KUKA KRL program: Machining2.src

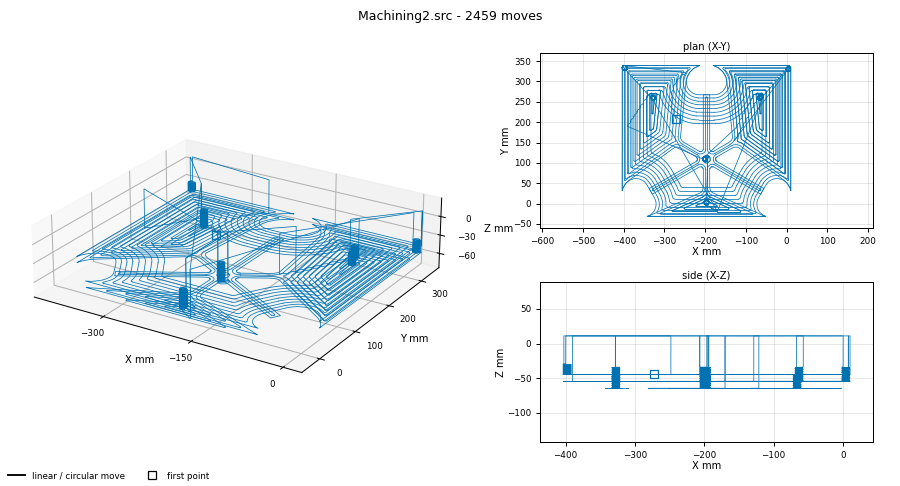
[picture p0: tool path of Machining2.src, 2459 of 2459 moves have a stored position in this frame; points joined in program order, loops and branches not executed]
&ACCESS RVP
&REL 1
&PARAM TEMPLATE = C:\KRC\Roboter\Template\vorgabe
&PARAM EDITMASK = *
DEF Machining2 ( )

; External program calls:
EXT Machining3()

CIRC {X -271.618,Y 203.851,Z -44.500,A 0.015,B -0.000,C -180.000},{X -272.375,Y 208.247,Z -44.500,A 0.015,B -0.000,C -180.000} C_DIS
CIRC {X -272.985,Y 212.625,Z -44.500,A 0.015,B 0.000,C 180.000},{X -275.736,Y 216.083,Z -44.500,A 0.015,B 0.000,C 180.000} C_DIS
CIRC {X -297.181,Y 237.599,Z -44.500,A 0.015,B -0.000,C 180.000},{X -311.042,Y 264.630,Z -44.500,A 0.015,B -0.000,C -180.000} C_DIS
CIRC {X -313.145,Y 267.504,Z -44.500,A 0.015,B 0.000,C 180.000},{X -316.534,Y 268.601,Z -44.500,A 0.015,B 0.000,C 180.000} C_DIS
LIN {X -329.332,Y 268.600,Z -44.500,A 0.015,B 0.000,C 180.000} C_DIS
CIRC {X -332.056,Y 267.472,Z -44.500,A 0.015,B 0.000,C -180.000},{X -333.185,Y 264.747,Z -44.500,A 0.015,B 0.000,C -180.000} C_DIS
LIN {X -333.181,Y 129.664,Z -44.500,A 0.015,B -0.000,C 180.000} C_DIS
CIRC {X -332.044,Y 125.846,Z -44.500,A 0.015,B 0.000,C 180.000},{X -329.005,Y 123.272,Z -44.500,A 0.015,B 0.000,C 180.000} C_DIS
CIRC {X -324.117,Y 121.053,Z -44.500,A 0.015,B 0.000,C 180.000},{X -319.285,Y 118.713,Z -44.500,A 0.015,B 0.000,C 180.000} C_DIS
CIRC {X -314.570,Y 116.140,Z -44.500,A 0.015,B 0.000,C -180.000},{X -310.050,Y 113.238,Z -44.500,A 0.015,B 0.000,C -180.000} C_DIS
CIRC {X -294.805,Y 99.946,Z -44.500,A 0.015,B 0.000,C -180.000},{X -282.838,Y 83.640,Z -44.500,A 0.015,B 0.000,C 180.000} C_DIS
LIN {X -263.188,Y 49.540,Z -44.500,A 0.015,B 0.000,C 180.000} C_DIS
CIRC {X -262.373,Y 48.033,Z -44.500,A 0.015,B 0.000,C 180.000},{X -261.642,Y 46.485,Z -44.500,A 0.015,B 0.000,C -180.000} C_DIS
CIRC {X -260.946,Y 44.921,Z -44.500,A 0.015,B 0.000,C 180.000},{X -260.238,Y 43.362,Z -44.500,A 0.015,B 0.000,C 180.000} C_DIS
CIRC {X -257.688,Y 40.428,Z -44.500,A 0.015,B 0.000,C -180.000},{X -253.958,Y 39.334,Z -44.500,A 0.015,B 0.000,C 180.000} C_DIS
LIN {X -139.525,Y 39.335,Z -44.500,A 0.015,B 0.000,C 180.000} C_DIS
CIRC {X -135.796,Y 40.433,Z -44.500,A 0.015,B -0.000,C -180.000},{X -133.257,Y 43.377,Z -44.500,A 0.015,B 0.000,C 180.000} C_DIS
CIRC {X -132.507,Y 45.047,Z -44.500,A 0.015,B 0.000,C 180.000},{X -131.768,Y 46.722,Z -44.500,A 0.015,B -0.000,C 180.000} C_DIS
CIRC {X -130.987,Y 48.379,Z -44.500,A 0.015,B 0.000,C -180.000},{X -130.115,Y 49.990,Z -44.500,A 0.015,B 0.000,C -180.000} C_DIS
LIN {X -109.644,Y 85.014,Z -44.500,A 0.015,B -0.000,C 180.000} C_DIS
CIRC {X -97.349,Y 101.310,Z -44.500,A 0.015,B 0.000,C 180.000},{X -81.729,Y 114.451,Z -44.500,A 0.015,B 0.000,C 180.000} C_DIS
CIRC {X -77.604,Y 116.999,Z -44.500,A 0.015,B 0.000,C 180.000},{X -73.317,Y 119.264,Z -44.500,A 0.015,B 0.000,C -180.000} C_DIS
CIRC {X -68.933,Y 121.328,Z -44.500,A 0.015,B 0.000,C -180.000},{X -64.497,Y 123.278,Z -44.500,A 0.015,B 0.000,C 180.000} C_DIS
CIRC {X -61.466,Y 125.799,Z -44.500,A 0.015,B 0.000,C 180.000},{X -60.330,Y 129.575,Z -44.500,A 0.015,B 0.000,C 180.000} C_DIS
LIN {X -60.333,Y 264.754,Z -44.500,A 0.015,B 0.000,C 180.000} C_DIS
CIRC {X -61.462,Y 267.478,Z -44.500,A 0.015,B 0.000,C 180.000},{X -64.186,Y 268.607,Z -44.500,A 0.015,B -0.000,C -180.000} C_DIS
LIN {X -76.977,Y 268.606,Z -44.500,A 0.015,B 0.000,C -180.000} C_DIS
CIRC {X -80.365,Y 267.510,Z -44.500,A 0.015,B 0.000,C 180.000},{X -82.468,Y 264.636,Z -44.500,A 0.015,B 0.000,C 180.000} C_DIS
CIRC {X -91.051,Y 245.836,Z -44.500,A 0.015,B 0.000,C -180.000},{X -103.514,Y 229.351,Z -44.500,A 0.015,B 0.000,C 180.000} C_DIS
CIRC {X -119.021,Y 215.739,Z -44.500,A 0.015,B -0.000,C -180.000},{X -136.787,Y 205.249,Z -44.500,A 0.015,B -0.000,C -180.000} C_DIS
CIRC {X -155.589,Y 198.757,Z -44.500,A 0.015,B 0.000,C 180.000},{X -175.343,Y 196.423,Z -44.500,A 0.015,B 0.000,C 180.000} C_DIS
LIN {X -214.895,Y 196.221,Z -44.500,A 0.015,B 0.000,C 180.000} C_DIS
CIRC {X -245.902,Y 200.993,Z -44.500,A 0.015,B 0.000,C 180.000},{X -274.038,Y 214.868,Z -44.500,A 0.015,B 0.000,C 180.000} C_DIS
CIRC {X -274.890,Y 215.471,Z -44.500,A 0.015,B 0.000,C 180.000},{X -275.736,Y 216.083,Z -44.500,A 0.015,B 0.000,C -180.000} C_DIS
CIRC {X -278.577,Y 219.932,Z -44.500,A 0.015,B 0.000,C 180.000},{X -278.721,Y 224.714,Z -44.500,A 0.015,B 0.000,C 180.000} C_DIS
CIRC {X -278.679,Y 229.444,Z -44.500,A 0.015,B 0.000,C 180.000},{X -281.022,Y 233.552,Z -44.500,A 0.015,B 0.000,C 180.000} C_DIS
CIRC {X -283.384,Y 236.013,Z -44.500,A 0.015,B 0.000,C -180.000},{X -285.659,Y 238.555,Z -44.500,A 0.015,B 0.000,C 180.000} C_DIS
CIRC {X -296.886,Y 255.155,Z -44.500,A 0.015,B 0.000,C 180.000},{X -303.914,Y 273.923,Z -44.500,A 0.015,B 0.000,C 180.000} C_DIS
CIRC {X -305.790,Y 276.833,Z -44.500,A 0.015,B 0.000,C -180.000},{X -309.063,Y 277.963,Z -44.500,A 0.015,B 0.000,C -180.000} C_DIS
LIN {X -338.695,Y 277.963,Z -44.500,A 0.015,B -0.000,C 180.000} C_DIS
CIRC {X -341.419,Y 276.834,Z -44.500,A 0.015,B -0.000,C -180.000},{X -342.547,Y 274.110,Z -44.500,A 0.015,B -0.000,C 180.000} C_DIS
LIN {X -342.543,Y 123.023,Z -44.500,A 0.015,B 0.000,C 180.000} C_DIS
CIRC {X -341.454,Y 119.492,Z -44.500,A 0.015,B 0.000,C 180.000},{X -338.566,Y 117.188,Z -44.500,A 0.015,B 0.000,C 180.000} C_DIS
CIRC {X -332.560,Y 114.714,Z -44.500,A 0.015,B 0.000,C 180.000},{X -326.639,Y 112.042,Z -44.500,A 0.015,B 0.000,C 180.000} C_DIS
CIRC {X -320.879,Y 109.028,Z -44.500,A 0.015,B 0.000,C -180.000},{X -315.388,Y 105.546,Z -44.500,A 0.015,B -0.000,C 180.000} C_DIS
CIRC {X -301.093,Y 93.048,Z -44.500,A 0.015,B 0.000,C -180.000},{X -289.921,Y 77.693,Z -44.500,A 0.015,B 0.000,C -180.000} C_DIS
LIN {X -271.167,Y 44.942,Z -44.500,A 0.015,B 0.000,C 180.000} C_DIS
CIRC {X -269.801,Y 42.329,Z -44.500,A 0.015,B 0.000,C 180.000},{X -268.653,Y 39.612,Z -44.500,A 0.015,B -0.000,C -180.000} C_DIS
CIRC {X -267.596,Y 36.862,Z -44.500,A 0.015,B 0.000,C 180.000},{X -266.491,Y 34.130,Z -44.500,A 0.015,B 0.000,C -180.000} C_DIS
CIRC {X -264.009,Y 31.107,Z -44.500,A 0.015,B 0.000,C 180.000},{X -260.265,Y 29.972,Z -44.500,A 0.015,B 0.000,C 180.000} C_DIS
LIN {X -133.256,Y 29.972,Z -44.500,A 0.015,B 0.000,C -180.000} C_DIS
CIRC {X -129.505,Y 31.106,Z -44.500,A 0.015,B -0.000,C -180.000},{X -127.010,Y 34.129,Z -44.500,A 0.015,B 0.000,C -180.000} C_DIS
CIRC {X -125.855,Y 36.970,Z -44.500,A 0.015,B 0.000,C 180.000},{X -124.756,Y 39.833,Z -44.500,A 0.015,B 0.000,C -180.000} C_DIS
CIRC {X -123.565,Y 42.662,Z -44.500,A 0.015,B 0.000,C -180.000},{X -122.142,Y 45.382,Z -44.500,A 0.015,B -0.000,C -180.000} C_DIS
LIN {X -103.037,Y 78.441,Z -44.500,A 0.015,B -0.000,C 180.000} C_DIS
CIRC {X -91.420,Y 94.078,Z -44.500,A 0.015,B 0.000,C 180.000},{X -76.544,Y 106.655,Z -44.500,A 0.015,B 0.000,C 180.000} C_DIS
CIRC {X -71.400,Y 109.776,Z -44.500,A 0.015,B 0.000,C 180.000},{X -66.016,Y 112.459,Z -44.500,A 0.015,B 0.000,C 180.000} C_DIS
CIRC {X -60.505,Y 114.859,Z -44.500,A 0.015,B 0.000,C -180.000},{X -54.946,Y 117.146,Z -44.500,A 0.015,B -0.000,C 180.000} C_DIS
CIRC {X -52.055,Y 119.473,Z -44.500,A 0.015,B 0.000,C -180.000},{X -50.967,Y 123.022,Z -44.500,A 0.015,B 0.000,C 180.000} C_DIS
LIN {X -50.971,Y 274.117,Z -44.500,A 0.015,B 0.000,C 180.000} C_DIS
CIRC {X -52.100,Y 276.841,Z -44.500,A 0.015,B 0.000,C -180.000},{X -54.824,Y 277.969,Z -44.500,A 0.015,B 0.000,C -180.000} C_DIS
LIN {X -84.496,Y 277.969,Z -44.500,A 0.015,B -0.000,C -180.000} C_DIS
CIRC {X -87.755,Y 276.836,Z -44.500,A 0.015,B 0.000,C -180.000},{X -89.608,Y 273.925,Z -44.500,A 0.015,B 0.000,C 180.000} C_DIS
CIRC {X -106.660,Y 239.262,Z -44.500,A 0.015,B -0.000,C -180.000},{X -137.083,Y 215.457,Z -44.500,A 0.015,B -0.000,C -180.000} C_DIS
CIRC {X -147.019,Y 211.354,Z -44.500,A 0.015,B -0.000,C -180.000},{X -157.305,Y 208.228,Z -44.500,A 0.015,B 0.000,C 180.000} C_DIS
CIRC {X -167.879,Y 206.247,Z -44.500,A 0.015,B 0.000,C -180.000},{X -178.617,Y 205.584,Z -44.500,A 0.015,B 0.000,C 180.000} C_DIS
LIN {X -216.069,Y 205.584,Z -44.500,A 0.015,B 0.000,C -180.000} C_DIS
CIRC {X -235.574,Y 207.795,Z -44.500,A 0.015,B 0.000,C -180.000},{X -254.089,Y 214.317,Z -44.500,A 0.015,B 0.000,C 180.000} C_DIS
CIRC {X -268.368,Y 222.797,Z -44.500,A 0.015,B -0.000,C -180.000},{X -281.022,Y 233.552,Z -44.500,A 0.015,B 0.000,C 180.000} C_DIS
CIRC {X -283.064,Y 237.540,Z -44.500,A 0.015,B 0.000,C -180.000},{X -282.419,Y 241.973,Z -44.500,A 0.015,B 0.000,C 180.000} C_DIS
CIRC {X -281.599,Y 246.322,Z -44.500,A 0.015,B -0.000,C 180.000},{X -283.108,Y 250.482,Z -44.500,A 0.015,B 0.000,C 180.000} C_DIS
CIRC {X -285.499,Y 254.008,Z -44.500,A 0.015,B -0.000,C -180.000},{X -287.754,Y 257.623,Z -44.500,A 0.015,B 0.000,C 180.000} C_DIS
CIRC {X -291.877,Y 265.858,Z -44.500,A 0.015,B 0.000,C 180.000},{X -294.729,Y 274.615,Z -44.500,A 0.015,B 0.000,C -180.000} C_DIS
CIRC {X -295.216,Y 276.775,Z -44.500,A 0.015,B 0.000,C 180.000},{X -295.626,Y 278.952,Z -44.500,A 0.015,B 0.000,C -180.000} C_DIS
CIRC {X -296.025,Y 281.130,Z -44.500,A 0.015,B -0.000,C 180.000},{X -296.480,Y 283.297,Z -44.500,A 0.015,B 0.000,C 180.000} C_DIS
CIRC {X -298.286,Y 286.195,Z -44.500,A 0.015,B 0.000,C -180.000},{X -301.508,Y 287.326,Z -44.500,A 0.015,B -0.000,C 180.000} C_DIS
LIN {X -348.057,Y 287.325,Z -44.500,A 0.015,B 0.000,C -180.000} C_DIS
CIRC {X -350.782,Y 286.196,Z -44.500,A 0.015,B 0.000,C 180.000},{X -351.910,Y 283.472,Z -44.500,A 0.015,B 0.000,C -180.000} C_DIS
LIN {X -351.906,Y 115.520,Z -44.500,A 0.015,B 0.000,C -180.000} C_DIS
CIRC {X -350.817,Y 112.320,Z -44.500,A 0.015,B 0.000,C -180.000},{X -348.003,Y 110.446,Z -44.500,A 0.015,B -0.000,C -180.000} C_DIS
CIRC {X -338.196,Y 107.179,Z -44.500,A 0.015,B 0.000,C 180.000},{X -328.868,Y 102.725,Z -44.500,A 0.015,B -0.000,C -180.000} C_DIS
CIRC {X -320.144,Y 97.184,Z -44.500,A 0.015,B 0.000,C -180.000},{X -312.124,Y 90.665,Z -44.500,A 0.015,B 0.000,C -180.000} C_DIS
CIRC {X -307.860,Y 86.416,Z -44.500,A 0.015,B 0.000,C -180.000},{X -303.971,Y 81.821,Z -44.500,A 0.015,B 0.000,C -180.000} C_DIS
CIRC {X -300.448,Y 76.943,Z -44.500,A 0.015,B 0.000,C -180.000},{X -297.267,Y 71.835,Z -44.500,A 0.015,B 0.000,C -180.000} C_DIS
LIN {X -283.335,Y 47.658,Z -44.500,A 0.015,B 0.000,C -180.000} C_DIS
CIRC {X -277.503,Y 36.349,Z -44.500,A 0.015,B 0.000,C -180.000},{X -272.749,Y 24.546,Z -44.500,A 0.015,B -0.000,C -180.000} C_DIS
CIRC {X -270.603,Y 21.694,Z -44.500,A 0.015,B 0.000,C -180.000},{X -267.203,Y 20.609,Z -44.500,A 0.015,B -0.000,C 180.000} C_DIS
LIN {X -126.309,Y 20.609,Z -44.500,A 0.015,B 0.000,C 180.000} C_DIS
CIRC {X -122.909,Y 21.694,Z -44.500,A 0.015,B 0.000,C -180.000},{X -120.763,Y 24.546,Z -44.500,A 0.015,B 0.000,C -180.000} C_DIS
CIRC {X -115.935,Y 36.521,Z -44.500,A 0.015,B -0.000,C -180.000},{X -110.007,Y 47.991,Z -44.500,A 0.015,B -0.000,C -180.000} C_DIS
LIN {X -96.029,Y 72.178,Z -44.500,A 0.015,B 0.000,C 180.000} C_DIS
CIRC {X -90.459,Y 80.530,Z -44.500,A 0.015,B -0.000,C -180.000},{X -83.866,Y 88.100,Z -44.500,A 0.015,B 0.000,C 180.000} C_DIS
CIRC {X -76.453,Y 94.859,Z -44.500,A 0.015,B 0.000,C 180.000},{X -68.393,Y 100.832,Z -44.500,A 0.015,B 0.000,C 180.000} C_DIS
CIRC {X -63.022,Y 103.997,Z -44.500,A 0.015,B 0.000,C -180.000},{X -57.338,Y 106.559,Z -44.500,A 0.015,B 0.000,C -180.000} C_DIS
CIRC {X -51.474,Y 108.656,Z -44.500,A 0.015,B 0.000,C 180.000},{X -45.510,Y 110.450,Z -44.500,A 0.015,B 0.000,C 180.000} C_DIS
CIRC {X -42.692,Y 112.346,Z -44.500,A 0.015,B 0.000,C 180.000},{X -41.604,Y 115.564,Z -44.500,A 0.015,B -0.000,C -180.000} C_DIS
LIN {X -41.609,Y 283.479,Z -44.500,A 0.015,B 0.000,C 180.000} C_DIS
CIRC {X -42.737,Y 286.204,Z -44.500,A 0.015,B 0.000,C 180.000},{X -45.462,Y 287.332,Z -44.500,A 0.015,B 0.000,C -180.000} C_DIS
LIN {X -91.945,Y 287.331,Z -44.500,A 0.015,B 0.000,C 180.000} C_DIS
CIRC {X -95.170,Y 286.210,Z -44.500,A 0.015,B 0.000,C -180.000},{X -97.004,Y 283.330,Z -44.500,A 0.015,B 0.000,C -180.000} C_DIS
LIN {X -99.842,Y 271.336,Z -44.500,A 0.015,B 0.000,C -180.000} C_DIS
CIRC {X -101.575,Y 265.775,Z -44.500,A 0.015,B 0.000,C -180.000},{X -104.064,Y 260.510,Z -44.500,A 0.015,B -0.000,C 180.000} C_DIS
CIRC {X -117.581,Y 242.142,Z -44.500,A 0.015,B -0.000,C -180.000},{X -135.162,Y 227.618,Z -44.500,A 0.015,B 0.000,C -180.000} C_DIS
CIRC {X -155.984,Y 218.179,Z -44.500,A 0.015,B 0.000,C 180.000},{X -178.617,Y 214.946,Z -44.500,A 0.015,B 0.000,C 180.000} C_DIS
LIN {X -222.088,Y 215.412,Z -44.500,A 0.015,B 0.000,C 180.000} C_DIS
CIRC {X -237.419,Y 218.560,Z -44.500,A 0.015,B -0.000,C 180.000},{X -252.126,Y 223.912,Z -44.500,A 0.015,B 0.000,C 180.000} C_DIS
CIRC {X -265.647,Y 231.902,Z -44.500,A 0.015,B 0.000,C 180.000},{X -277.069,Y 242.683,Z -44.500,A 0.015,B -0.000,C 180.000} C_DIS
CIRC {X -280.174,Y 246.516,Z -44.500,A 0.015,B 0.000,C 180.000},{X -283.108,Y 250.482,Z -44.500,A 0.015,B -0.000,C -180.000} C_DIS
CIRC {X -284.531,Y 254.910,Z -44.500,A 0.015,B 0.000,C -180.000},{X -283.170,Y 259.358,Z -44.500,A 0.015,B 0.000,C -180.000} C_DIS
CIRC {X -281.622,Y 263.677,Z -44.500,A 0.015,B 0.000,C -180.000},{X -282.392,Y 268.200,Z -44.500,A 0.015,B 0.000,C -180.000} C_DIS
CIRC {X -284.981,Y 274.803,Z -44.500,A 0.015,B 0.000,C -180.000},{X -286.881,Y 281.636,Z -44.500,A 0.015,B 0.000,C -180.000} C_DIS
CIRC {X -287.971,Y 287.239,Z -44.500,A 0.015,B -0.000,C -180.000},{X -288.752,Y 292.893,Z -44.500,A 0.015,B -0.000,C -180.000} C_DIS
CIRC {X -290.148,Y 295.601,Z -44.500,A 0.015,B -0.000,C 180.000},{X -292.995,Y 296.689,Z -44.500,A 0.015,B 0.000,C 180.000} C_DIS
LIN {X -357.420,Y 296.687,Z -44.500,A 0.015,B 0.000,C 180.000} C_DIS
CIRC {X -360.145,Y 295.559,Z -44.500,A 0.015,B -0.000,C 180.000},{X -361.273,Y 292.834,Z -44.500,A 0.015,B -0.000,C 180.000} C_DIS
LIN {X -361.268,Y 107.604,Z -44.500,A 0.015,B 0.000,C 180.000} C_DIS
CIRC {X -360.139,Y 104.482,Z -44.500,A 0.015,B 0.000,C -180.000},{X -357.273,Y 102.804,Z -44.500,A 0.015,B -0.000,C -180.000} C_DIS
LIN {X -350.128,Y 101.484,Z -44.500,A 0.015,B -0.000,C 180.000} C_DIS
CIRC {X -346.790,Y 100.665,Z -44.500,A 0.015,B 0.000,C -180.000},{X -343.568,Y 99.468,Z -44.500,A 0.015,B 0.000,C -180.000} C_DIS
CIRC {X -332.303,Y 93.624,Z -44.500,A 0.015,B 0.000,C -180.000},{X -321.890,Y 86.369,Z -44.500,A 0.015,B -0.000,C 180.000} C_DIS
CIRC {X -312.732,Y 77.539,Z -44.500,A 0.015,B -0.000,C 180.000},{X -305.379,Y 67.160,Z -44.500,A 0.015,B 0.000,C 180.000} C_DIS
CIRC {X -298.046,Y 54.649,Z -44.500,A 0.015,B -0.000,C -180.000},{X -290.530,Y 42.247,Z -44.500,A 0.015,B 0.000,C -180.000} C_DIS
CIRC {X -284.018,Y 29.227,Z -44.500,A 0.015,B 0.000,C -180.000},{X -279.898,Y 15.264,Z -44.500,A 0.015,B -0.000,C 180.000} C_DIS
CIRC {X -278.163,Y 12.379,Z -44.500,A 0.015,B 0.000,C 180.000},{X -274.992,Y 11.247,Z -44.500,A 0.015,B -0.000,C 180.000} C_DIS
LIN {X -118.588,Y 11.247,Z -44.500,A 0.015,B 0.000,C -180.000} C_DIS
CIRC {X -115.391,Y 12.378,Z -44.500,A 0.015,B -0.000,C -180.000},{X -113.618,Y 15.268,Z -44.500,A 0.015,B 0.000,C 180.000} C_DIS
CIRC {X -112.298,Y 20.666,Z -44.500,A 0.015,B 0.000,C 180.000},{X -110.662,Y 25.977,Z -44.500,A 0.015,B 0.000,C 180.000} C_DIS
CIRC {X -108.613,Y 31.148,Z -44.500,A 0.015,B -0.000,C -180.000},{X -106.069,Y 36.093,Z -44.500,A 0.015,B 0.000,C 180.000} C_DIS
LIN {X -84.511,Y 72.588,Z -44.500,A 0.015,B 0.000,C -180.000} C_DIS
CIRC {X -75.252,Y 82.913,Z -44.500,A 0.015,B -0.000,C 180.000},{X -64.558,Y 91.742,Z -44.500,A 0.015,B 0.000,C 180.000} C_DIS
CIRC {X -52.386,Y 98.481,Z -44.500,A 0.015,B 0.000,C 180.000},{X -39.039,Y 102.410,Z -44.500,A 0.015,B -0.000,C 180.000} C_DIS
CIRC {X -38.340,Y 102.523,Z -44.500,A 0.015,B 0.000,C 180.000},{X -37.638,Y 102.615,Z -44.500,A 0.015,B 0.000,C 180.000} C_DIS
CIRC {X -36.936,Y 102.707,Z -44.500,A 0.015,B -0.000,C -180.000},{X -36.237,Y 102.820,Z -44.500,A 0.015,B 0.000,C 180.000} C_DIS
CIRC {X -33.372,Y 104.480,Z -44.500,A 0.015,B -0.000,C 180.000},{X -32.241,Y 107.593,Z -44.500,A 0.015,B 0.000,C 180.000} C_DIS
LIN {X -32.246,Y 292.842,Z -44.500,A 0.015,B 0.000,C -180.000} C_DIS
CIRC {X -33.375,Y 295.567,Z -44.500,A 0.015,B 0.000,C 180.000},{X -36.099,Y 296.695,Z -44.500,A 0.015,B -0.000,C -180.000} C_DIS
LIN {X -100.551,Y 296.694,Z -44.500,A 0.015,B 0.000,C 180.000} C_DIS
CIRC {X -103.382,Y 295.606,Z -44.500,A 0.015,B -0.000,C 180.000},{X -104.755,Y 292.902,Z -44.500,A 0.015,B 0.000,C -180.000} C_DIS
CIRC {X -106.056,Y 284.390,Z -44.500,A 0.015,B 0.000,C 180.000},{X -108.180,Y 276.046,Z -44.500,A 0.015,B 0.000,C -180.000} C_DIS
CIRC {X -111.145,Y 267.960,Z -44.500,A 0.015,B -0.000,C -180.000},{X -114.954,Y 260.236,Z -44.500,A 0.015,B -0.000,C -180.000} C_DIS
CIRC {X -122.919,Y 249.060,Z -44.500,A 0.015,B 0.000,C 180.000},{X -133.090,Y 239.846,Z -44.500,A 0.015,B 0.000,C -180.000} C_DIS
CIRC {X -144.761,Y 232.696,Z -44.500,A 0.015,B -0.000,C -180.000},{X -157.409,Y 227.466,Z -44.500,A 0.015,B 0.000,C 180.000} C_DIS
CIRC {X -162.596,Y 226.032,Z -44.500,A 0.015,B 0.000,C 180.000},{X -167.889,Y 225.055,Z -44.500,A 0.015,B 0.000,C 180.000} C_DIS
CIRC {X -173.240,Y 224.496,Z -44.500,A 0.015,B -0.000,C 180.000},{X -178.617,Y 224.309,Z -44.500,A 0.015,B -0.000,C -180.000} C_DIS
LIN {X -220.881,Y 224.696,Z -44.500,A 0.015,B 0.000,C 180.000} C_DIS
CIRC {X -234.529,Y 227.465,Z -44.500,A 0.015,B 0.000,C -180.000},{X -247.649,Y 232.135,Z -44.500,A 0.015,B 0.000,C -180.000} C_DIS
CIRC {X -259.735,Y 239.162,Z -44.500,A 0.015,B 0.000,C -180.000},{X -269.925,Y 248.735,Z -44.500,A 0.015,B 0.000,C -180.000} C_DIS
CIRC {X -275.572,Y 256.167,Z -44.500,A 0.015,B -0.000,C 180.000},{X -280.400,Y 264.156,Z -44.500,A 0.015,B 0.000,C 180.000} C_DIS
CIRC {X -281.429,Y 266.162,Z -44.500,A 0.015,B 0.000,C -180.000},{X -282.392,Y 268.200,Z -44.500,A 0.015,B 0.000,C -180.000} C_DIS
CIRC {X -282.943,Y 272.549,Z -44.500,A 0.015,B -0.000,C -180.000},{X -280.949,Y 276.452,Z -44.500,A 0.015,B -0.000,C 180.000} C_DIS
CIRC {X -278.767,Y 280.173,Z -44.500,A 0.015,B 0.000,C -180.000},{X -278.560,Y 284.481,Z -44.500,A 0.015,B -0.000,C -180.000} C_DIS
CIRC {X -278.662,Y 285.023,Z -44.500,A 0.015,B 0.000,C -180.000},{X -278.759,Y 285.566,Z -44.500,A 0.015,B 0.000,C 180.000} C_DIS
CIRC {X -279.645,Y 293.969,Z -44.500,A 0.015,B 0.000,C 180.000},{X -279.424,Y 302.416,Z -44.500,A 0.015,B 0.000,C -180.000} C_DIS
CIRC {X -280.280,Y 304.966,Z -44.500,A 0.015,B 0.000,C 180.000},{X -282.740,Y 306.052,Z -44.500,A 0.015,B 0.000,C 180.000} C_DIS
LIN {X -366.783,Y 306.050,Z -44.500,A 0.015,B -0.000,C -180.000} C_DIS
CIRC {X -369.508,Y 304.921,Z -44.500,A 0.015,B 0.000,C 180.000},{X -370.636,Y 302.197,Z -44.500,A 0.015,B 0.000,C -180.000} C_DIS
LIN {X -370.630,Y 98.481,Z -44.500,A 0.015,B 0.000,C -180.000} C_DIS
CIRC {X -369.542,Y 95.797,Z -44.500,A 0.015,B -0.000,C -180.000},{X -366.892,Y 94.628,Z -44.500,A 0.015,B 0.000,C 180.000} C_DIS
CIRC {X -355.317,Y 93.164,Z -44.500,A 0.015,B 0.000,C 180.000},{X -344.232,Y 89.522,Z -44.500,A 0.015,B 0.000,C 180.000} C_DIS
CIRC {X -333.977,Y 83.985,Z -44.500,A 0.015,B -0.000,C -180.000},{X -324.764,Y 76.849,Z -44.500,A 0.015,B 0.000,C -180.000} C_DIS
CIRC {X -321.522,Y 73.611,Z -44.500,A 0.015,B 0.000,C 180.000},{X -318.575,Y 70.101,Z -44.500,A 0.015,B -0.000,C 180.000} C_DIS
CIRC {X -315.908,Y 66.377,Z -44.500,A 0.015,B 0.000,C 180.000},{X -313.491,Y 62.485,Z -44.500,A 0.015,B 0.000,C 180.000} C_DIS
LIN {X -293.225,Y 26.693,Z -44.500,A 0.015,B 0.000,C 180.000} C_DIS
CIRC {X -291.298,Y 21.603,Z -44.500,A 0.015,B 0.000,C 180.000},{X -289.690,Y 16.404,Z -44.500,A 0.015,B 0.000,C -180.000} C_DIS
CIRC {X -288.476,Y 11.096,Z -44.500,A 0.015,B 0.000,C 180.000},{X -287.735,Y 5.702,Z -44.500,A 0.015,B 0.000,C 180.000} C_DIS
CIRC {X -286.381,Y 2.982,Z -44.500,A 0.015,B -0.000,C -180.000},{X -283.548,Y 1.884,Z -44.500,A 0.015,B 0.000,C -180.000} C_DIS
LIN {X -110.014,Y 1.884,Z -44.500,A 0.015,B -0.000,C 180.000} C_DIS
CIRC {X -107.106,Y 3.014,Z -44.500,A 0.015,B 0.000,C 180.000},{X -105.725,Y 5.812,Z -44.500,A 0.015,B 0.000,C 180.000} C_DIS
CIRC {X -104.809,Y 12.484,Z -44.500,A 0.015,B 0.000,C 180.000},{X -103.246,Y 19.035,Z -44.500,A 0.015,B 0.000,C 180.000} C_DIS
CIRC {X -100.977,Y 25.381,Z -44.500,A 0.015,B 0.000,C 180.000},{X -97.963,Y 31.408,Z -44.500,A 0.015,B 0.000,C 180.000} C_DIS
LIN {X -77.092,Y 66.876,Z -44.500,A 0.015,B 0.000,C 180.000} C_DIS
CIRC {X -69.013,Y 75.975,Z -44.500,A 0.015,B 0.000,C 180.000},{X -59.744,Y 83.859,Z -44.500,A 0.015,B 0.000,C 180.000} C_DIS
CIRC {X -49.143,Y 89.933,Z -44.500,A 0.015,B 0.000,C -180.000},{X -37.439,Y 93.440,Z -44.500,A 0.015,B -0.000,C -180.000} C_DIS
CIRC {X -34.750,Y 93.878,Z -44.500,A 0.015,B 0.000,C 180.000},{X -32.049,Y 94.233,Z -44.500,A 0.015,B -0.000,C -180.000} C_DIS
CIRC {X -29.337,Y 94.489,Z -44.500,A 0.015,B 0.000,C -180.000},{X -26.616,Y 94.628,Z -44.500,A 0.015,B -0.000,C 180.000} C_DIS
CIRC {X -23.966,Y 95.797,Z -44.500,A 0.015,B 0.000,C 180.000},{X -22.878,Y 98.480,Z -44.500,A 0.015,B -0.000,C 180.000} C_DIS
LIN {X -22.884,Y 302.205,Z -44.500,A 0.015,B 0.000,C 180.000} C_DIS
CIRC {X -24.013,Y 304.930,Z -44.500,A 0.015,B 0.000,C 180.000},{X -26.737,Y 306.058,Z -44.500,A 0.015,B 0.000,C 180.000} C_DIS
LIN {X -110.808,Y 306.056,Z -44.500,A 0.015,B -0.000,C 180.000} C_DIS
CIRC {X -113.254,Y 304.962,Z -44.500,A 0.015,B 0.000,C 180.000},{X -114.068,Y 302.410,Z -44.500,A 0.015,B 0.000,C 180.000} C_DIS
CIRC {X -115.316,Y 282.677,Z -44.500,A 0.015,B 0.000,C -180.000},{X -123.245,Y 264.565,Z -44.500,A 0.015,B 0.000,C -180.000} C_DIS
CIRC {X -136.251,Y 249.834,Z -44.500,A 0.015,B 0.000,C -180.000},{X -152.735,Y 239.134,Z -44.500,A 0.015,B 0.000,C 180.000} C_DIS
CIRC {X -157.806,Y 237.117,Z -44.500,A 0.015,B 0.000,C 180.000},{X -163.086,Y 235.736,Z -44.500,A 0.015,B 0.000,C -180.000} C_DIS
CIRC {X -168.447,Y 234.771,Z -44.500,A 0.015,B 0.000,C 180.000},{X -173.837,Y 233.981,Z -44.500,A 0.015,B 0.000,C 180.000} C_DIS
LIN {X -214.895,Y 233.671,Z -44.500,A 0.015,B -0.000,C -180.000} C_DIS
CIRC {X -232.628,Y 236.252,Z -44.500,A 0.015,B -0.000,C 180.000},{X -248.889,Y 243.778,Z -44.500,A 0.015,B -0.000,C 180.000} C_DIS
CIRC {X -262.570,Y 255.261,Z -44.500,A 0.015,B 0.000,C -180.000},{X -273.119,Y 269.675,Z -44.500,A 0.015,B 0.000,C -180.000} C_DIS
CIRC {X -276.430,Y 276.861,Z -44.500,A 0.015,B 0.000,C 180.000},{X -278.560,Y 284.481,Z -44.500,A 0.015,B -0.000,C 180.000} C_DIS
CIRC {X -278.095,Y 288.859,Z -44.500,A 0.015,B 0.000,C 180.000},{X -275.248,Y 292.218,Z -44.500,A 0.015,B 0.000,C 180.000} C_DIS
CIRC {X -272.244,Y 295.330,Z -44.500,A 0.015,B 0.000,C -180.000},{X -270.968,Y 299.464,Z -44.500,A 0.015,B 0.000,C -180.000} C_DIS
LIN {X -270.899,Y 300.374,Z -44.500,A 0.015,B -0.000,C -180.000} C_DIS
CIRC {X -270.563,Y 303.151,Z -44.500,A 0.015,B 0.000,C -180.000},{X -270.037,Y 305.900,Z -44.500,A 0.015,B 0.000,C 180.000} C_DIS
CIRC {X -269.466,Y 308.637,Z -44.500,A 0.015,B 0.000,C 180.000},{X -268.994,Y 311.394,Z -44.500,A 0.015,B 0.000,C 180.000} C_DIS
CIRC {X -269.727,Y 313.957,Z -44.500,A 0.015,B -0.000,C 180.000},{X -272.150,Y 315.070,Z -44.500,A 0.015,B 0.000,C -180.000} C_DIS
LIN {X -375.801,Y 315.067,Z -44.500,A 0.015,B 0.000,C 180.000} C_DIS
CIRC {X -378.526,Y 313.939,Z -44.500,A 0.015,B -0.000,C -180.000},{X -379.654,Y 311.214,Z -44.500,A 0.015,B 0.000,C 180.000} C_DIS
LIN {X -379.648,Y 88.694,Z -44.500,A 0.015,B -0.000,C -180.000} C_DIS
CIRC {X -378.574,Y 86.266,Z -44.500,A 0.015,B 0.000,C -180.000},{X -376.054,Y 85.427,Z -44.500,A 0.015,B 0.000,C 180.000} C_DIS
CIRC {X -355.378,Y 83.757,Z -44.500,A 0.015,B -0.000,C 180.000},{X -336.545,Y 75.062,Z -44.500,A 0.015,B 0.000,C 180.000} C_DIS
CIRC {X -332.723,Y 72.022,Z -44.500,A 0.015,B 0.000,C 180.000},{X -329.330,Y 68.509,Z -44.500,A 0.015,B -0.000,C -180.000} C_DIS
CIRC {X -326.231,Y 64.747,Z -44.500,A 0.015,B 0.000,C 180.000},{X -323.238,Y 60.901,Z -44.500,A 0.015,B -0.000,C -180.000} C_DIS
LIN {X -303.164,Y 26.503,Z -44.500,A 0.015,B 0.000,C 180.000} C_DIS
CIRC {X -297.523,Y 12.024,Z -44.500,A 0.015,B -0.000,C 180.000},{X -296.453,Y -3.479,Z -44.500,A 0.015,B -0.000,C 180.000} C_DIS
CIRC {X -295.565,Y -6.045,Z -44.500,A 0.015,B 0.000,C 180.000},{X -293.078,Y -7.134,Z -44.500,A 0.015,B -0.000,C 180.000} C_DIS
LIN {X -100.409,Y -7.134,Z -44.500,A 0.015,B -0.000,C 180.000} C_DIS
CIRC {X -97.912,Y -6.032,Z -44.500,A 0.015,B -0.000,C -180.000},{X -97.044,Y -3.446,Z -44.500,A 0.015,B 0.000,C -180.000} C_DIS
CIRC {X -97.116,Y 3.540,Z -44.500,A 0.015,B 0.000,C 180.000},{X -96.058,Y 10.445,Z -44.500,A 0.015,B 0.000,C 180.000} C_DIS
CIRC {X -94.171,Y 17.153,Z -44.500,A 0.015,B 0.000,C -180.000},{X -91.746,Y 23.686,Z -44.500,A 0.015,B 0.000,C 180.000} C_DIS
LIN {X -72.009,Y 58.296,Z -44.500,A 0.015,B 0.000,C 180.000} C_DIS
CIRC {X -61.990,Y 70.842,Z -44.500,A 0.015,B 0.000,C -180.000},{X -48.714,Y 79.870,Z -44.500,A 0.015,B 0.000,C -180.000} C_DIS
CIRC {X -33.464,Y 84.783,Z -44.500,A 0.015,B 0.000,C 180.000},{X -17.454,Y 85.427,Z -44.500,A 0.015,B 0.000,C 180.000} C_DIS
CIRC {X -14.935,Y 86.265,Z -44.500,A 0.015,B 0.000,C -180.000},{X -13.860,Y 88.693,Z -44.500,A 0.015,B 0.000,C -180.000} C_DIS
LIN {X -13.866,Y 311.223,Z -44.500,A 0.015,B -0.000,C -180.000} C_DIS
CIRC {X -14.995,Y 313.948,Z -44.500,A 0.015,B 0.000,C 180.000},{X -17.719,Y 315.076,Z -44.500,A 0.015,B -0.000,C 180.000} C_DIS
LIN {X -121.362,Y 315.074,Z -44.500,A 0.015,B 0.000,C -180.000} C_DIS
CIRC {X -123.765,Y 313.973,Z -44.500,A 0.015,B 0.000,C -180.000},{X -124.501,Y 311.435,Z -44.500,A 0.015,B 0.000,C 180.000} C_DIS
CIRC {X -123.710,Y 306.391,Z -44.500,A 0.015,B 0.000,C 180.000},{X -122.837,Y 301.361,Z -44.500,A 0.015,B 0.000,C 180.000} C_DIS
CIRC {X -122.442,Y 296.244,Z -44.500,A 0.015,B -0.000,C 180.000},{X -123.104,Y 291.154,Z -44.500,A 0.015,B 0.000,C 180.000} C_DIS
CIRC {X -124.909,Y 284.207,Z -44.500,A 0.015,B 0.000,C -180.000},{X -127.017,Y 277.345,Z -44.500,A 0.015,B 0.000,C 180.000} C_DIS
CIRC {X -129.929,Y 270.749,Z -44.500,A 0.015,B 0.000,C 180.000},{X -134.042,Y 264.828,Z -44.500,A 0.015,B -0.000,C 180.000} C_DIS
CIRC {X -141.130,Y 257.492,Z -44.500,A 0.015,B -0.000,C 180.000},{X -149.112,Y 251.142,Z -44.500,A 0.015,B 0.000,C -180.000} C_DIS
CIRC {X -158.171,Y 246.342,Z -44.500,A 0.015,B -0.000,C -180.000},{X -168.107,Y 243.819,Z -44.500,A 0.015,B -0.000,C -180.000} C_DIS
CIRC {X -170.727,Y 243.465,Z -44.500,A 0.015,B 0.000,C -180.000},{X -173.343,Y 243.085,Z -44.500,A 0.015,B -0.000,C 180.000} C_DIS
CIRC {X -175.973,Y 242.788,Z -44.500,A 0.015,B 0.000,C 180.000},{X -178.617,Y 242.689,Z -44.500,A 0.015,B 0.000,C -180.000} C_DIS
LIN {X -218.512,Y 242.923,Z -44.500,A 0.015,B -0.000,C -180.000} C_DIS
CIRC {X -228.857,Y 244.948,Z -44.500,A 0.015,B -0.000,C -180.000},{X -238.859,Y 248.277,Z -44.500,A 0.015,B 0.000,C 180.000} C_DIS
CIRC {X -248.128,Y 253.414,Z -44.500,A 0.015,B 0.000,C -180.000},{X -255.901,Y 260.616,Z -44.500,A 0.015,B 0.000,C -180.000} C_DIS
CIRC {X -262.304,Y 269.390,Z -44.500,A 0.015,B 0.000,C 180.000},{X -267.373,Y 278.996,Z -44.500,A 0.015,B 0.000,C 180.000} C_DIS
CIRC {X -270.400,Y 289.014,Z -44.500,A 0.015,B 0.000,C 180.000},{X -270.968,Y 299.464,Z -44.500,A 0.015,B 0.000,C -180.000} C_DIS
CIRC {X -269.461,Y 303.549,Z -44.500,A 0.015,B 0.000,C 180.000},{X -265.971,Y 306.153,Z -44.500,A 0.015,B 0.000,C -180.000} C_DIS
CIRC {X -262.396,Y 308.526,Z -44.500,A 0.015,B 0.000,C 180.000},{X -260.266,Y 312.251,Z -44.500,A 0.015,B 0.000,C -180.000} C_DIS
CIRC {X -258.787,Y 316.418,Z -44.500,A 0.015,B -0.000,C 180.000},{X -256.861,Y 320.398,Z -44.500,A 0.015,B 0.000,C -180.000} C_DIS
CIRC {X -256.892,Y 322.649,Z -44.500,A 0.015,B 0.000,C 180.000},{X -258.847,Y 323.765,Z -44.500,A 0.015,B -0.000,C 180.000} C_DIS
LIN {X -384.497,Y 323.762,Z -44.500,A 0.015,B -0.000,C -180.000} C_DIS
CIRC {X -387.221,Y 322.634,Z -44.500,A 0.015,B 0.000,C -180.000},{X -388.349,Y 319.909,Z -44.500,A 0.015,B 0.000,C 180.000} C_DIS
LIN {X -388.343,Y 76.974,Z -44.500,A 0.015,B 0.000,C -180.000} C_DIS
CIRC {X -387.221,Y 74.738,Z -44.500,A 0.015,B 0.000,C 180.000},{X -384.758,Y 74.301,Z -44.500,A 0.015,B 0.000,C 180.000} C_DIS
CIRC {X -382.026,Y 75.170,Z -44.500,A 0.015,B 0.000,C 180.000},{X -379.328,Y 76.138,Z -44.500,A 0.015,B -0.000,C 180.000} C_DIS
CIRC {X -376.559,Y 76.921,Z -44.500,A 0.015,B 0.000,C 180.000},{X -373.697,Y 77.211,Z -44.500,A 0.015,B -0.000,C -180.000} C_DIS
CIRC {X -364.547,Y 76.724,Z -44.500,A 0.015,B 0.000,C 180.000},{X -355.543,Y 75.022,Z -44.500,A 0.015,B 0.000,C -180.000} C_DIS
CIRC {X -346.974,Y 71.644,Z -44.500,A 0.015,B 0.000,C 180.000},{X -339.472,Y 66.298,Z -44.500,A 0.015,B 0.000,C -180.000} C_DIS
CIRC {X -336.490,Y 63.417,Z -44.500,A 0.015,B 0.000,C -180.000},{X -333.669,Y 60.379,Z -44.500,A 0.015,B -0.000,C -180.000} C_DIS
CIRC {X -331.086,Y 57.130,Z -44.500,A 0.015,B 0.000,C 180.000},{X -328.838,Y 53.642,Z -44.500,A 0.015,B 0.000,C 180.000} C_DIS
LIN {X -309.588,Y 19.910,Z -44.500,A 0.015,B 0.000,C -180.000} C_DIS
CIRC {X -307.470,Y 14.262,Z -44.500,A 0.015,B 0.000,C 180.000},{X -305.744,Y 8.483,Z -44.500,A 0.015,B 0.000,C -180.000} C_DIS
CIRC {X -304.765,Y 2.509,Z -44.500,A 0.015,B -0.000,C 180.000},{X -304.914,Y -3.543,Z -44.500,A 0.015,B -0.000,C -180.000} C_DIS
CIRC {X -305.197,Y -5.765,Z -44.500,A 0.015,B 0.000,C -180.000},{X -305.516,Y -7.982,Z -44.500,A 0.015,B 0.000,C 180.000} C_DIS
CIRC {X -305.895,Y -10.190,Z -44.500,A 0.015,B 0.000,C 180.000},{X -306.354,Y -12.382,Z -44.500,A 0.015,B 0.000,C 180.000} C_DIS
CIRC {X -305.811,Y -14.767,Z -44.500,A 0.015,B 0.000,C 180.000},{X -303.607,Y -15.829,Z -44.500,A 0.015,B -0.000,C 180.000} C_DIS
LIN {X -89.904,Y -15.829,Z -44.500,A 0.015,B 0.000,C -180.000} C_DIS
CIRC {X -87.701,Y -14.767,Z -44.500,A 0.015,B 0.000,C 180.000},{X -87.158,Y -12.382,Z -44.500,A 0.015,B -0.000,C -180.000} C_DIS
CIRC {X -88.156,Y -6.743,Z -44.500,A 0.015,B 0.000,C 180.000},{X -88.589,Y -1.034,Z -44.500,A 0.015,B -0.000,C -180.000} C_DIS
CIRC {X -88.399,Y 4.692,Z -44.500,A 0.015,B 0.000,C -180.000},{X -87.536,Y 10.356,Z -44.500,A 0.015,B 0.000,C -180.000} C_DIS
CIRC {X -86.696,Y 13.546,Z -44.500,A 0.015,B 0.000,C 180.000},{X -85.560,Y 16.644,Z -44.500,A 0.015,B 0.000,C -180.000} C_DIS
CIRC {X -84.186,Y 19.641,Z -44.500,A 0.015,B 0.000,C -180.000},{X -82.627,Y 22.546,Z -44.500,A 0.015,B 0.000,C 180.000} C_DIS
LIN {X -63.058,Y 56.070,Z -44.500,A 0.015,B 0.000,C 180.000} C_DIS
CIRC {X -53.476,Y 66.044,Z -44.500,A 0.015,B 0.000,C 180.000},{X -41.961,Y 73.705,Z -44.500,A 0.015,B -0.000,C 180.000} C_DIS
CIRC {X -28.518,Y 77.644,Z -44.500,A 0.015,B 0.000,C 180.000},{X -14.581,Y 76.238,Z -44.500,A 0.015,B 0.000,C -180.000} C_DIS
CIRC {X -13.115,Y 75.770,Z -44.500,A 0.015,B -0.000,C 180.000},{X -11.663,Y 75.256,Z -44.500,A 0.015,B 0.000,C -180.000} C_DIS
CIRC {X -10.212,Y 74.742,Z -44.500,A 0.015,B 0.000,C 180.000},{X -8.746,Y 74.274,Z -44.500,A 0.015,B -0.000,C -180.000} C_DIS
CIRC {X -6.287,Y 74.703,Z -44.500,A 0.015,B 0.000,C -180.000},{X -5.165,Y 76.934,Z -44.500,A 0.015,B -0.000,C 180.000} C_DIS
LIN {X -5.172,Y 319.918,Z -44.500,A 0.015,B 0.000,C 180.000} C_DIS
CIRC {X -6.300,Y 322.643,Z -44.500,A 0.015,B -0.000,C 180.000},{X -9.025,Y 323.771,Z -44.500,A 0.015,B 0.000,C 180.000} C_DIS
LIN {X -134.603,Y 323.768,Z -44.500,A 0.015,B 0.000,C -180.000} C_DIS
CIRC {X -136.588,Y 322.651,Z -44.500,A 0.015,B 0.000,C -180.000},{X -136.663,Y 320.374,Z -44.500,A 0.015,B 0.000,C -180.000} C_DIS
CIRC {X -133.781,Y 313.945,Z -44.500,A 0.015,B 0.000,C 180.000},{X -131.666,Y 307.224,Z -44.500,A 0.015,B -0.000,C -180.000} C_DIS
CIRC {X -130.769,Y 300.196,Z -44.500,A 0.015,B 0.000,C -180.000},{X -131.565,Y 293.156,Z -44.500,A 0.015,B 0.000,C 180.000} C_DIS
CIRC {X -133.884,Y 284.868,Z -44.500,A 0.015,B 0.000,C 180.000},{X -136.867,Y 276.795,Z -44.500,A 0.015,B 0.000,C -180.000} C_DIS
CIRC {X -141.242,Y 269.301,Z -44.500,A 0.015,B -0.000,C -180.000},{X -147.443,Y 263.231,Z -44.500,A 0.015,B -0.000,C 180.000} C_DIS
CIRC {X -154.510,Y 258.580,Z -44.500,A 0.015,B -0.000,C -180.000},{X -162.073,Y 254.789,Z -44.500,A 0.015,B 0.000,C 180.000} C_DIS
CIRC {X -170.171,Y 252.244,Z -44.500,A 0.015,B 0.000,C -180.000},{X -178.617,Y 251.384,Z -44.500,A 0.015,B 0.000,C 180.000} C_DIS
LIN {X -217.391,Y 251.546,Z -44.500,A 0.015,B 0.000,C -180.000} C_DIS
CIRC {X -226.175,Y 253.219,Z -44.500,A 0.015,B 0.000,C -180.000},{X -234.701,Y 255.914,Z -44.500,A 0.015,B -0.000,C -180.000} C_DIS
CIRC {X -242.636,Y 260.155,Z -44.500,A 0.015,B -0.000,C 180.000},{X -249.267,Y 266.236,Z -44.500,A 0.015,B 0.000,C -180.000} C_DIS
CIRC {X -252.981,Y 271.048,Z -44.500,A 0.015,B 0.000,C -180.000},{X -256.243,Y 276.176,Z -44.500,A 0.015,B 0.000,C -180.000} C_DIS
CIRC {X -258.868,Y 281.671,Z -44.500,A 0.015,B -0.000,C 180.000},{X -260.638,Y 287.497,Z -44.500,A 0.015,B 0.000,C 180.000} C_DIS
CIRC {X -261.844,Y 295.852,Z -44.500,A 0.015,B 0.000,C 180.000},{X -261.765,Y 304.294,Z -44.500,A 0.015,B 0.000,C -180.000} C_DIS
CIRC {X -261.215,Y 308.310,Z -44.500,A 0.015,B 0.000,C -180.000},{X -260.266,Y 312.251,Z -44.500,A 0.015,B 0.000,C -180.000} C_DIS
CIRC {X -258.078,Y 315.414,Z -44.500,A 0.015,B 0.000,C -180.000},{X -254.437,Y 316.654,Z -44.500,A 0.015,B 0.000,C 180.000} C_DIS
CIRC {X -250.793,Y 317.660,Z -44.500,A 0.015,B 0.000,C 180.000},{X -248.130,Y 320.342,Z -44.500,A 0.015,B 0.000,C -180.000} C_DIS
CIRC {X -247.435,Y 321.545,Z -44.500,A 0.015,B 0.000,C -180.000},{X -246.733,Y 322.745,Z -44.500,A 0.015,B 0.000,C 180.000} C_DIS
CIRC {X -244.610,Y 325.939,Z -44.500,A 0.015,B 0.000,C -180.000},{X -242.147,Y 328.880,Z -44.500,A 0.015,B 0.000,C -180.000} C_DIS
CIRC {X -241.814,Y 330.800,Z -44.500,A 0.015,B 0.000,C 180.000},{X -243.443,Y 331.870,Z -44.500,A 0.015,B -0.000,C 180.000} C_DIS
LIN {X -392.601,Y 331.866,Z -44.500,A 0.015,B 0.000,C -180.000} C_DIS
CIRC {X -395.325,Y 330.738,Z -44.500,A 0.015,B -0.000,C -180.000},{X -396.454,Y 328.013,Z -44.500,A 0.015,B -0.000,C -180.000} C_DIS
LIN {X -396.447,Y 62.472,Z -44.500,A 0.015,B 0.000,C -180.000} C_DIS
CIRC {X -395.334,Y 60.698,Z -44.500,A 0.015,B 0.000,C 180.000},{X -393.254,Y 60.927,Z -44.500,A 0.015,B 0.000,C -180.000} C_DIS
CIRC {X -391.495,Y 62.327,Z -44.500,A 0.015,B 0.000,C -180.000},{X -389.744,Y 63.738,Z -44.500,A 0.015,B -0.000,C 180.000} C_DIS
CIRC {X -387.858,Y 64.982,Z -44.500,A 0.015,B -0.000,C -180.000},{X -385.767,Y 65.835,Z -44.500,A 0.015,B 0.000,C -180.000} C_DIS
LIN {X -376.055,Y 68.685,Z -44.500,A 0.015,B 0.000,C 180.000} C_DIS
CIRC {X -371.030,Y 69.523,Z -44.500,A 0.015,B 0.000,C 180.000},{X -365.947,Y 69.183,Z -44.500,A 0.015,B -0.000,C 180.000} C_DIS
CIRC {X -358.950,Y 67.502,Z -44.500,A 0.015,B 0.000,C 180.000},{X -352.172,Y 65.089,Z -44.500,A 0.015,B -0.000,C -180.000} C_DIS
CIRC {X -345.907,Y 61.442,Z -44.500,A 0.015,B 0.000,C 180.000},{X -340.812,Y 56.287,Z -44.500,A 0.015,B 0.000,C 180.000} C_DIS
CIRC {X -339.538,Y 54.639,Z -44.500,A 0.015,B 0.000,C 180.000},{X -338.231,Y 53.018,Z -44.500,A 0.015,B 0.000,C 180.000} C_DIS
CIRC {X -336.974,Y 51.356,Z -44.500,A 0.015,B -0.000,C 180.000},{X -335.860,Y 49.595,Z -44.500,A 0.015,B 0.000,C -180.000} C_DIS
LIN {X -317.074,Y 16.806,Z -44.500,A 0.015,B 0.000,C 180.000} C_DIS
CIRC {X -314.647,Y 9.864,Z -44.500,A 0.015,B 0.000,C -180.000},{X -313.018,Y 2.692,Z -44.500,A 0.015,B 0.000,C 180.000} C_DIS
CIRC {X -312.736,Y -4.706,Z -44.500,A 0.015,B 0.000,C -180.000},{X -314.344,Y -11.933,Z -44.500,A 0.015,B -0.000,C 180.000} C_DIS
CIRC {X -315.200,Y -14.162,Z -44.500,A 0.015,B -0.000,C -180.000},{X -316.138,Y -16.358,Z -44.500,A 0.015,B -0.000,C 180.000} C_DIS
CIRC {X -317.178,Y -18.509,Z -44.500,A 0.015,B -0.000,C 180.000},{X -318.337,Y -20.597,Z -44.500,A 0.015,B -0.000,C 180.000} C_DIS
CIRC {X -318.357,Y -22.817,Z -44.500,A 0.015,B 0.000,C -180.000},{X -316.437,Y -23.933,Z -44.500,A 0.015,B 0.000,C -180.000} C_DIS
LIN {X -77.107,Y -23.933,Z -44.500,A 0.015,B 0.000,C 180.000} C_DIS
CIRC {X -75.172,Y -22.817,Z -44.500,A 0.015,B 0.000,C -180.000},{X -75.171,Y -20.584,Z -44.500,A 0.015,B 0.000,C -180.000} C_DIS
CIRC {X -77.636,Y -15.754,Z -44.500,A 0.015,B 0.000,C 180.000},{X -79.602,Y -10.699,Z -44.500,A 0.015,B 0.000,C 180.000} C_DIS
CIRC {X -80.782,Y -5.384,Z -44.500,A 0.015,B 0.000,C -180.000},{X -80.860,Y 0.060,Z -44.500,A 0.015,B 0.000,C -180.000} C_DIS
CIRC {X -80.244,Y 4.844,Z -44.500,A 0.015,B 0.000,C 180.000},{X -79.244,Y 9.563,Z -44.500,A 0.015,B 0.000,C 180.000} C_DIS
CIRC {X -77.734,Y 14.152,Z -44.500,A 0.015,B 0.000,C 180.000},{X -75.610,Y 18.491,Z -44.500,A 0.015,B 0.000,C 180.000} C_DIS
LIN {X -56.636,Y 51.126,Z -44.500,A 0.015,B 0.000,C -180.000} C_DIS
CIRC {X -51.793,Y 56.776,Z -44.500,A 0.015,B -0.000,C -180.000},{X -46.383,Y 61.887,Z -44.500,A 0.015,B 0.000,C 180.000} C_DIS
CIRC {X -40.082,Y 65.948,Z -44.500,A 0.015,B 0.000,C -180.000},{X -32.939,Y 68.225,Z -44.500,A 0.015,B 0.000,C -180.000} C_DIS
CIRC {X -25.143,Y 69.092,Z -44.500,A 0.015,B 0.000,C 180.000},{X -17.300,Y 68.927,Z -44.500,A 0.015,B 0.000,C -180.000} C_DIS
CIRC {X -9.603,Y 67.089,Z -44.500,A 0.015,B -0.000,C -180.000},{X -2.775,Y 63.089,Z -44.500,A 0.015,B -0.000,C 180.000} C_DIS
CIRC {X -2.134,Y 62.556,Z -44.500,A 0.015,B 0.000,C -180.000},{X -1.510,Y 62.004,Z -44.500,A 0.015,B -0.000,C -180.000} C_DIS
CIRC {X -0.886,Y 61.452,Z -44.500,A 0.015,B 0.000,C 180.000},{X -0.245,Y 60.919,Z -44.500,A 0.015,B -0.000,C -180.000} C_DIS
CIRC {X 1.828,Y 60.679,Z -44.500,A 0.015,B 0.000,C 180.000},{X 2.940,Y 62.444,Z -44.500,A 0.015,B 0.000,C -180.000} C_DIS
LIN {X 2.932,Y 328.023,Z -44.500,A 0.015,B 0.000,C 180.000} C_DIS
CIRC {X 1.804,Y 330.747,Z -44.500,A 0.015,B 0.000,C 180.000},{X -0.921,Y 331.876,Z -44.500,A 0.015,B 0.000,C -180.000} C_DIS
LIN {X -150.071,Y 331.872,Z -44.500,A 0.015,B 0.000,C -180.000} C_DIS
CIRC {X -151.701,Y 330.802,Z -44.500,A 0.015,B 0.000,C 180.000},{X -151.367,Y 328.882,Z -44.500,A 0.015,B 0.000,C -180.000} C_DIS
CIRC {X -146.021,Y 321.988,Z -44.500,A 0.015,B 0.000,C 180.000},{X -142.045,Y 314.223,Z -44.500,A 0.015,B 0.000,C 180.000} C_DIS
CIRC {X -139.686,Y 305.811,Z -44.500,A 0.015,B 0.000,C 180.000},{X -139.161,Y 297.091,Z -44.500,A 0.015,B 0.000,C 180.000} C_DIS
CIRC {X -141.737,Y 285.043,Z -44.500,A 0.015,B 0.000,C -180.000},{X -148.060,Y 274.469,Z -44.500,A 0.015,B 0.000,C -180.000} C_DIS
CIRC {X -157.213,Y 266.292,Z -44.500,A 0.015,B -0.000,C 180.000},{X -168.253,Y 260.933,Z -44.500,A 0.015,B 0.000,C -180.000} C_DIS
CIRC {X -170.788,Y 260.244,Z -44.500,A 0.015,B 0.000,C -180.000},{X -173.378,Y 259.804,Z -44.500,A 0.015,B 0.000,C -180.000} C_DIS
CIRC {X -175.993,Y 259.567,Z -44.500,A 0.015,B -0.000,C 180.000},{X -178.617,Y 259.488,Z -44.500,A 0.015,B -0.000,C 180.000} C_DIS
LIN {X -216.347,Y 259.582,Z -44.500,A 0.015,B 0.000,C 180.000} C_DIS
CIRC {X -223.676,Y 260.928,Z -44.500,A 0.015,B 0.000,C 180.000},{X -230.826,Y 263.031,Z -44.500,A 0.015,B 0.000,C 180.000} C_DIS
CIRC {X -237.517,Y 266.437,Z -44.500,A 0.015,B -0.000,C -180.000},{X -243.083,Y 271.475,Z -44.500,A 0.015,B 0.000,C -180.000} C_DIS
CIRC {X -246.212,Y 275.503,Z -44.500,A 0.015,B -0.000,C 180.000},{X -248.986,Y 279.784,Z -44.500,A 0.015,B 0.000,C 180.000} C_DIS
CIRC {X -251.229,Y 284.377,Z -44.500,A 0.015,B -0.000,C 180.000},{X -252.729,Y 289.263,Z -44.500,A 0.015,B 0.000,C -180.000} C_DIS
CIRC {X -253.818,Y 296.030,Z -44.500,A 0.015,B -0.000,C -180.000},{X -254.087,Y 302.879,Z -44.500,A 0.015,B -0.000,C 180.000} C_DIS
CIRC {X -253.111,Y 309.702,Z -44.500,A 0.015,B 0.000,C -180.000},{X -250.528,Y 316.091,Z -44.500,A 0.015,B -0.000,C -180.000} C_DIS
CIRC {X -249.338,Y 318.222,Z -44.500,A 0.015,B 0.000,C -180.000},{X -248.130,Y 320.342,Z -44.500,A 0.015,B 0.000,C 180.000} C_DIS
LIN {X -247.972,Y 320.950,Z -44.330,A 0.015,B -0.000,C 180.000} C_DIS
LIN {X -248.053,Y 321.405,Z -43.865,A 0.015,B -0.000,C -180.000} C_DIS
LIN {X -248.124,Y 321.560,Z -43.230,A 0.015,B 0.000,C 180.000} C_DIS
$VEL.CP = 1.00000
LIN {X -248.124,Y 321.560,Z 11.000,A 0.015,B -0.000,C -180.000} C_DIS
$VEL.CP = 1.00000
LIN {X -399.689,Y 339.077,Z 11.000,A 0.015,B 0.000,C 180.000} C_DIS
$VEL.CP = 0.10000
LIN {X -399.689,Y 339.077,Z -28.231,A 0.015,B 0.000,C -180.000} C_DIS
LIN {X -399.692,Y 339.076,Z -28.330,A 0.015,B 0.000,C -180.000} C_DIS
LIN {X -399.828,Y 339.053,Z -28.813,A 0.015,B 0.000,C -180.000} C_DIS
LIN {X -400.133,Y 338.983,Z -29.204,A 0.015,B 0.000,C -180.000} C_DIS
LIN {X -400.552,Y 338.848,Z -29.444,A 0.015,B -0.000,C -180.000} C_DIS
LIN {X -400.596,Y 338.832,Z -29.458,A 0.015,B 0.000,C -180.000} C_DIS
LIN {X -400.858,Y 338.722,Z -29.500,A 0.015,B 0.000,C 180.000} C_DIS
LIN {X -401.281,Y 338.494,Z -29.517,A 0.015,B 0.000,C 180.000} C_DIS
LIN {X -401.404,Y 338.418,Z -29.522,A 0.015,B 0.000,C 180.000} C_DIS
LIN {X -402.842,Y 337.053,Z -29.592,A 0.015,B 0.000,C 180.000} C_DIS
LIN {X -402.866,Y 337.018,Z -29.593,A 0.015,B 0.000,C -180.000} C_DIS
LIN {X -403.753,Y 334.430,Z -29.690,A 0.015,B -0.000,C -180.000} C_DIS
LIN {X -403.779,Y 333.946,Z -29.707,A 0.015,B -0.000,C -180.000} C_DIS
LIN {X -403.787,Y 333.653,Z -29.717,A 0.015,B -0.000,C -180.000} C_DIS
LIN {X -403.787,Y 333.050,Z -29.738,A 0.015,B 0.000,C -180.000} C_DIS
LIN {X -401.252,Y 328.076,Z -29.940,A 0.015,B 0.000,C -180.000} C_DIS
LIN {X -395.738,Y 327.203,Z -30.143,A 0.015,B -0.000,C -180.000} C_DIS
LIN {X -391.790,Y 331.150,Z -30.345,A 0.015,B 0.000,C -180.000} C_DIS
LIN {X -392.664,Y 336.664,Z -30.548,A 0.015,B -0.000,C -180.000} C_DIS
LIN {X -397.638,Y 339.199,Z -30.750,A 0.015,B -0.000,C -180.000} C_DIS
LIN {X -398.507,Y 339.199,Z -30.780,A 0.015,B -0.000,C -180.000} C_DIS
LIN {X -399.336,Y 339.133,Z -30.809,A 0.015,B 0.000,C 180.000} C_DIS
LIN {X -399.692,Y 339.076,Z -30.822,A 0.015,B 0.000,C -180.000} C_DIS
LIN {X -400.552,Y 338.848,Z -30.853,A 0.015,B 0.000,C -180.000} C_DIS
LIN {X -400.596,Y 338.832,Z -30.855,A 0.015,B -0.000,C -180.000} C_DIS
LIN {X -401.281,Y 338.494,Z -30.881,A 0.015,B 0.000,C -180.000} C_DIS
LIN {X -401.404,Y 338.418,Z -30.886,A 0.015,B -0.000,C -180.000} C_DIS
LIN {X -402.842,Y 337.053,Z -30.956,A 0.015,B 0.000,C -180.000} C_DIS
LIN {X -402.866,Y 337.018,Z -30.958,A 0.015,B -0.000,C -180.000} C_DIS
LIN {X -403.753,Y 334.430,Z -31.054,A 0.015,B -0.000,C 180.000} C_DIS
LIN {X -403.779,Y 333.946,Z -31.071,A 0.015,B -0.000,C -180.000} C_DIS
LIN {X -403.787,Y 333.653,Z -31.082,A 0.015,B 0.000,C 180.000} C_DIS
LIN {X -403.787,Y 333.050,Z -31.103,A 0.015,B -0.000,C 180.000} C_DIS
LIN {X -401.252,Y 328.076,Z -31.305,A 0.015,B 0.000,C -180.000} C_DIS
LIN {X -395.738,Y 327.203,Z -31.507,A 0.015,B 0.000,C 180.000} C_DIS
LIN {X -391.790,Y 331.150,Z -31.710,A 0.015,B 0.000,C 180.000} C_DIS
LIN {X -392.664,Y 336.664,Z -31.912,A 0.015,B -0.000,C 180.000} C_DIS
LIN {X -397.638,Y 339.199,Z -32.114,A 0.015,B -0.000,C -180.000} C_DIS
LIN {X -398.507,Y 339.199,Z -32.145,A 0.015,B 0.000,C -180.000} C_DIS
LIN {X -399.336,Y 339.133,Z -32.174,A 0.015,B -0.000,C -180.000} C_DIS
LIN {X -399.692,Y 339.076,Z -32.186,A 0.015,B 0.000,C 180.000} C_DIS
LIN {X -400.552,Y 338.848,Z -32.218,A 0.015,B 0.000,C 180.000} C_DIS
LIN {X -400.596,Y 338.832,Z -32.219,A 0.015,B -0.000,C -180.000} C_DIS
LIN {X -401.281,Y 338.494,Z -32.246,A 0.015,B 0.000,C 180.000} C_DIS
LIN {X -401.404,Y 338.418,Z -32.251,A 0.015,B 0.000,C -180.000} C_DIS
LIN {X -402.842,Y 337.053,Z -32.321,A 0.015,B -0.000,C -180.000} C_DIS
LIN {X -402.866,Y 337.018,Z -32.322,A 0.015,B 0.000,C -180.000} C_DIS
LIN {X -403.753,Y 334.430,Z -32.419,A 0.015,B 0.000,C -180.000} C_DIS
LIN {X -403.779,Y 333.946,Z -32.436,A 0.015,B -0.000,C -180.000} C_DIS
LIN {X -403.787,Y 333.653,Z -32.446,A 0.015,B 0.000,C -180.000} C_DIS
LIN {X -403.787,Y 333.050,Z -32.467,A 0.015,B -0.000,C -180.000} C_DIS
LIN {X -401.252,Y 328.076,Z -32.669,A 0.015,B -0.000,C -180.000} C_DIS
LIN {X -395.738,Y 327.203,Z -32.872,A 0.015,B -0.000,C 180.000} C_DIS
LIN {X -391.790,Y 331.150,Z -33.074,A 0.015,B -0.000,C -180.000} C_DIS
LIN {X -392.664,Y 336.664,Z -33.277,A 0.015,B 0.000,C -180.000} C_DIS
LIN {X -397.638,Y 339.199,Z -33.479,A 0.015,B 0.000,C -180.000} C_DIS
LIN {X -398.507,Y 339.199,Z -33.509,A 0.015,B 0.000,C -180.000} C_DIS
LIN {X -399.336,Y 339.133,Z -33.538,A 0.015,B -0.000,C -180.000} C_DIS
LIN {X -399.692,Y 339.076,Z -33.551,A 0.015,B 0.000,C -180.000} C_DIS
LIN {X -400.552,Y 338.848,Z -33.582,A 0.015,B 0.000,C -180.000} C_DIS
LIN {X -400.596,Y 338.832,Z -33.584,A 0.015,B -0.000,C -180.000} C_DIS
LIN {X -401.281,Y 338.494,Z -33.610,A 0.015,B 0.000,C -180.000} C_DIS
LIN {X -401.404,Y 338.418,Z -33.615,A 0.015,B -0.000,C -180.000} C_DIS
LIN {X -402.842,Y 337.053,Z -33.685,A 0.015,B 0.000,C 180.000} C_DIS
LIN {X -402.866,Y 337.018,Z -33.687,A 0.015,B 0.000,C -180.000} C_DIS
LIN {X -403.753,Y 334.430,Z -33.783,A 0.015,B 0.000,C -180.000} C_DIS
LIN {X -403.779,Y 333.946,Z -33.800,A 0.015,B 0.000,C 180.000} C_DIS
LIN {X -403.787,Y 333.653,Z -33.811,A 0.015,B 0.000,C -180.000} C_DIS
LIN {X -403.787,Y 333.050,Z -33.832,A 0.015,B -0.000,C -180.000} C_DIS
LIN {X -401.252,Y 328.076,Z -34.034,A 0.015,B 0.000,C 180.000} C_DIS
LIN {X -395.738,Y 327.203,Z -34.236,A 0.015,B -0.000,C -180.000} C_DIS
LIN {X -391.790,Y 331.150,Z -34.439,A 0.015,B 0.000,C -180.000} C_DIS
LIN {X -392.664,Y 336.664,Z -34.641,A 0.015,B -0.000,C -180.000} C_DIS
LIN {X -397.638,Y 339.199,Z -34.843,A 0.015,B 0.000,C -180.000} C_DIS
LIN {X -398.507,Y 339.199,Z -34.874,A 0.015,B -0.000,C 180.000} C_DIS
LIN {X -399.336,Y 339.133,Z -34.903,A 0.015,B 0.000,C -180.000} C_DIS
LIN {X -399.692,Y 339.076,Z -34.915,A 0.015,B -0.000,C -180.000} C_DIS
LIN {X -400.552,Y 338.848,Z -34.947,A 0.015,B 0.000,C -180.000} C_DIS
LIN {X -400.596,Y 338.832,Z -34.948,A 0.015,B -0.000,C -180.000} C_DIS
LIN {X -401.281,Y 338.494,Z -34.975,A 0.015,B 0.000,C 180.000} C_DIS
LIN {X -401.404,Y 338.418,Z -34.980,A 0.015,B 0.000,C -180.000} C_DIS
LIN {X -402.842,Y 337.053,Z -35.050,A 0.015,B 0.000,C -180.000} C_DIS
LIN {X -402.866,Y 337.018,Z -35.051,A 0.015,B -0.000,C -180.000} C_DIS
LIN {X -403.753,Y 334.430,Z -35.148,A 0.015,B 0.000,C -180.000} C_DIS
LIN {X -403.779,Y 333.946,Z -35.165,A 0.015,B 0.000,C 180.000} C_DIS
LIN {X -403.787,Y 333.653,Z -35.175,A 0.015,B -0.000,C 180.000} C_DIS
LIN {X -403.787,Y 333.050,Z -35.196,A 0.015,B -0.000,C -180.000} C_DIS
LIN {X -401.252,Y 328.076,Z -35.399,A 0.015,B 0.000,C -180.000} C_DIS
LIN {X -395.738,Y 327.203,Z -35.601,A 0.015,B -0.000,C -180.000} C_DIS
LIN {X -391.790,Y 331.150,Z -35.803,A 0.015,B 0.000,C -180.000} C_DIS
LIN {X -392.664,Y 336.664,Z -36.006,A 0.015,B -0.000,C -180.000} C_DIS
LIN {X -397.638,Y 339.199,Z -36.208,A 0.015,B 0.000,C 180.000} C_DIS
LIN {X -398.507,Y 339.199,Z -36.238,A 0.015,B 0.000,C -180.000} C_DIS
LIN {X -399.336,Y 339.133,Z -36.267,A 0.015,B 0.000,C 180.000} C_DIS
LIN {X -399.692,Y 339.076,Z -36.280,A 0.015,B 0.000,C 180.000} C_DIS
LIN {X -400.552,Y 338.848,Z -36.311,A 0.015,B 0.000,C 180.000} C_DIS
LIN {X -400.596,Y 338.832,Z -36.313,A 0.015,B -0.000,C 180.000} C_DIS
LIN {X -401.281,Y 338.494,Z -36.339,A 0.015,B 0.000,C -180.000} C_DIS
LIN {X -401.404,Y 338.418,Z -36.345,A 0.015,B -0.000,C -180.000} C_DIS
LIN {X -402.842,Y 337.053,Z -36.414,A 0.015,B 0.000,C -180.000} C_DIS
LIN {X -402.866,Y 337.018,Z -36.416,A 0.015,B 0.000,C -180.000} C_DIS
LIN {X -403.753,Y 334.430,Z -36.513,A 0.015,B -0.000,C -180.000} C_DIS
LIN {X -403.779,Y 333.946,Z -36.529,A 0.015,B -0.000,C -180.000} C_DIS
LIN {X -403.787,Y 333.653,Z -36.540,A 0.015,B 0.000,C -180.000} C_DIS
LIN {X -403.787,Y 333.050,Z -36.561,A 0.015,B -0.000,C -180.000} C_DIS
LIN {X -401.252,Y 328.076,Z -36.763,A 0.015,B 0.000,C 180.000} C_DIS
LIN {X -395.738,Y 327.203,Z -36.965,A 0.015,B -0.000,C -180.000} C_DIS
LIN {X -391.790,Y 331.150,Z -37.168,A 0.015,B -0.000,C -180.000} C_DIS
LIN {X -392.664,Y 336.664,Z -37.370,A 0.015,B -0.000,C 180.000} C_DIS
LIN {X -397.638,Y 339.199,Z -37.573,A 0.015,B 0.000,C -180.000} C_DIS
LIN {X -398.507,Y 339.199,Z -37.603,A 0.015,B 0.000,C 180.000} C_DIS
LIN {X -399.336,Y 339.133,Z -37.632,A 0.015,B 0.000,C -180.000} C_DIS
LIN {X -399.692,Y 339.076,Z -37.645,A 0.015,B 0.000,C 180.000} C_DIS
LIN {X -400.552,Y 338.848,Z -37.676,A 0.015,B 0.000,C 180.000} C_DIS
LIN {X -400.596,Y 338.832,Z -37.677,A 0.015,B -0.000,C -180.000} C_DIS
LIN {X -401.281,Y 338.494,Z -37.704,A 0.015,B -0.000,C 180.000} C_DIS
LIN {X -401.404,Y 338.418,Z -37.709,A 0.015,B 0.000,C -180.000} C_DIS
LIN {X -402.842,Y 337.053,Z -37.779,A 0.015,B 0.000,C -180.000} C_DIS
LIN {X -402.866,Y 337.018,Z -37.780,A 0.015,B 0.000,C -180.000} C_DIS
LIN {X -403.753,Y 334.430,Z -37.877,A 0.015,B 0.000,C -180.000} C_DIS
LIN {X -403.779,Y 333.946,Z -37.894,A 0.015,B -0.000,C -180.000} C_DIS
LIN {X -403.787,Y 333.653,Z -37.904,A 0.015,B 0.000,C 180.000} C_DIS
LIN {X -403.787,Y 333.050,Z -37.925,A 0.015,B -0.000,C -180.000} C_DIS
LIN {X -401.252,Y 328.076,Z -38.128,A 0.015,B -0.000,C -180.000} C_DIS
LIN {X -395.738,Y 327.203,Z -38.330,A 0.015,B 0.000,C -180.000} C_DIS
LIN {X -391.790,Y 331.150,Z -38.532,A 0.015,B 0.000,C 180.000} C_DIS
LIN {X -392.664,Y 336.664,Z -38.735,A 0.015,B -0.000,C 180.000} C_DIS
LIN {X -397.638,Y 339.199,Z -38.937,A 0.015,B -0.000,C 180.000} C_DIS
LIN {X -398.507,Y 339.199,Z -38.967,A 0.015,B -0.000,C -180.000} C_DIS
LIN {X -399.336,Y 339.133,Z -38.996,A 0.015,B -0.000,C 180.000} C_DIS
LIN {X -399.692,Y 339.076,Z -39.009,A 0.015,B 0.000,C -180.000} C_DIS
LIN {X -400.552,Y 338.848,Z -39.040,A 0.015,B -0.000,C -180.000} C_DIS
LIN {X -400.596,Y 338.832,Z -39.042,A 0.015,B 0.000,C 180.000} C_DIS
LIN {X -401.281,Y 338.494,Z -39.069,A 0.015,B 0.000,C 180.000} C_DIS
LIN {X -401.404,Y 338.418,Z -39.074,A 0.015,B -0.000,C 180.000} C_DIS
LIN {X -402.842,Y 337.053,Z -39.143,A 0.015,B -0.000,C 180.000} C_DIS
LIN {X -402.866,Y 337.018,Z -39.145,A 0.015,B 0.000,C 180.000} C_DIS
LIN {X -403.753,Y 334.430,Z -39.242,A 0.015,B 0.000,C 180.000} C_DIS
LIN {X -403.779,Y 333.946,Z -39.259,A 0.015,B 0.000,C 180.000} C_DIS
LIN {X -403.787,Y 333.653,Z -39.269,A 0.015,B -0.000,C 180.000} C_DIS
LIN {X -403.787,Y 333.050,Z -39.290,A 0.015,B -0.000,C 180.000} C_DIS
LIN {X -401.252,Y 328.076,Z -39.492,A 0.015,B 0.000,C 180.000} C_DIS
LIN {X -395.738,Y 327.203,Z -39.695,A 0.015,B -0.000,C 180.000} C_DIS
LIN {X -391.790,Y 331.150,Z -39.897,A 0.015,B -0.000,C -180.000} C_DIS
LIN {X -392.664,Y 336.664,Z -40.099,A 0.015,B 0.000,C -180.000} C_DIS
LIN {X -397.638,Y 339.199,Z -40.302,A 0.015,B 0.000,C -180.000} C_DIS
LIN {X -398.507,Y 339.199,Z -40.332,A 0.015,B 0.000,C -180.000} C_DIS
LIN {X -399.336,Y 339.133,Z -40.361,A 0.015,B -0.000,C -180.000} C_DIS
LIN {X -399.692,Y 339.076,Z -40.374,A 0.015,B -0.000,C 180.000} C_DIS
LIN {X -400.552,Y 338.848,Z -40.405,A 0.015,B 0.000,C 180.000} C_DIS
LIN {X -400.596,Y 338.832,Z -40.406,A 0.015,B 0.000,C 180.000} C_DIS
LIN {X -401.281,Y 338.494,Z -40.433,A 0.015,B 0.000,C 180.000} C_DIS
LIN {X -401.404,Y 338.418,Z -40.438,A 0.015,B 0.000,C -180.000} C_DIS
LIN {X -402.842,Y 337.053,Z -40.508,A 0.015,B 0.000,C -180.000} C_DIS
LIN {X -402.866,Y 337.018,Z -40.509,A 0.015,B 0.000,C -180.000} C_DIS
LIN {X -403.753,Y 334.430,Z -40.606,A 0.015,B -0.000,C -180.000} C_DIS
LIN {X -403.779,Y 333.946,Z -40.623,A 0.015,B 0.000,C -180.000} C_DIS
LIN {X -403.787,Y 333.653,Z -40.633,A 0.015,B -0.000,C 180.000} C_DIS
LIN {X -403.787,Y 333.050,Z -40.654,A 0.015,B 0.000,C -180.000} C_DIS
LIN {X -401.252,Y 328.076,Z -40.857,A 0.015,B 0.000,C 180.000} C_DIS
LIN {X -395.738,Y 327.203,Z -41.059,A 0.015,B 0.000,C 180.000} C_DIS
LIN {X -391.790,Y 331.150,Z -41.261,A 0.015,B 0.000,C 180.000} C_DIS
LIN {X -392.664,Y 336.664,Z -41.464,A 0.015,B 0.000,C -180.000} C_DIS
LIN {X -397.638,Y 339.199,Z -41.666,A 0.015,B -0.000,C 180.000} C_DIS
LIN {X -398.507,Y 339.199,Z -41.696,A 0.015,B 0.000,C -180.000} C_DIS
LIN {X -399.336,Y 339.133,Z -41.726,A 0.015,B 0.000,C -180.000} C_DIS
LIN {X -399.692,Y 339.076,Z -41.738,A 0.015,B 0.000,C -180.000} C_DIS
LIN {X -400.552,Y 338.848,Z -41.769,A 0.015,B 0.000,C 180.000} C_DIS
LIN {X -400.596,Y 338.832,Z -41.771,A 0.015,B 0.000,C -180.000} C_DIS
LIN {X -401.281,Y 338.494,Z -41.798,A 0.015,B -0.000,C 180.000} C_DIS
LIN {X -401.404,Y 338.418,Z -41.803,A 0.015,B 0.000,C -180.000} C_DIS
LIN {X -402.842,Y 337.053,Z -41.872,A 0.015,B -0.000,C 180.000} C_DIS
LIN {X -402.866,Y 337.018,Z -41.874,A 0.015,B 0.000,C 180.000} C_DIS
LIN {X -403.753,Y 334.430,Z -41.971,A 0.015,B 0.000,C 180.000} C_DIS
LIN {X -403.779,Y 333.946,Z -41.988,A 0.015,B 0.000,C -180.000} C_DIS
LIN {X -403.787,Y 333.653,Z -41.998,A 0.015,B 0.000,C -180.000} C_DIS
LIN {X -403.787,Y 333.050,Z -42.019,A 0.015,B -0.000,C -180.000} C_DIS
LIN {X -401.252,Y 328.076,Z -42.221,A 0.015,B 0.000,C 180.000} C_DIS
LIN {X -395.738,Y 327.203,Z -42.424,A 0.015,B 0.000,C -180.000} C_DIS
LIN {X -391.790,Y 331.150,Z -42.626,A 0.015,B -0.000,C -180.000} C_DIS
LIN {X -392.664,Y 336.664,Z -42.828,A 0.015,B 0.000,C 180.000} C_DIS
LIN {X -397.638,Y 339.199,Z -43.031,A 0.015,B 0.000,C -180.000} C_DIS
LIN {X -398.507,Y 339.199,Z -43.061,A 0.015,B -0.000,C -180.000} C_DIS
LIN {X -399.336,Y 339.133,Z -43.090,A 0.015,B -0.000,C 180.000} C_DIS
LIN {X -399.692,Y 339.076,Z -43.103,A 0.015,B 0.000,C 180.000} C_DIS
LIN {X -400.552,Y 338.848,Z -43.134,A 0.015,B 0.000,C -180.000} C_DIS
LIN {X -400.596,Y 338.832,Z -43.135,A 0.015,B 0.000,C -180.000} C_DIS
LIN {X -401.281,Y 338.494,Z -43.162,A 0.015,B -0.000,C -180.000} C_DIS
LIN {X -401.404,Y 338.418,Z -43.167,A 0.015,B 0.000,C 180.000} C_DIS
LIN {X -402.842,Y 337.053,Z -43.237,A 0.015,B 0.000,C -180.000} C_DIS
LIN {X -402.866,Y 337.018,Z -43.238,A 0.015,B -0.000,C -180.000} C_DIS
LIN {X -403.753,Y 334.430,Z -43.335,A 0.015,B 0.000,C 180.000} C_DIS
LIN {X -403.779,Y 333.946,Z -43.352,A 0.015,B -0.000,C -180.000} C_DIS
LIN {X -403.787,Y 333.653,Z -43.362,A 0.015,B -0.000,C -180.000} C_DIS
LIN {X -403.787,Y 333.050,Z -43.383,A 0.015,B -0.000,C -180.000} C_DIS
LIN {X -401.252,Y 328.076,Z -43.586,A 0.015,B -0.000,C -180.000} C_DIS
LIN {X -395.738,Y 327.203,Z -43.788,A 0.015,B -0.000,C -180.000} C_DIS
LIN {X -391.790,Y 331.150,Z -43.991,A 0.015,B -0.000,C -180.000} C_DIS
LIN {X -392.664,Y 336.664,Z -44.193,A 0.015,B -0.000,C -180.000} C_DIS
LIN {X -397.638,Y 339.199,Z -44.395,A 0.015,B 0.000,C -180.000} C_DIS
LIN {X -398.507,Y 339.199,Z -44.426,A 0.015,B 0.000,C -180.000} C_DIS
LIN {X -399.336,Y 339.133,Z -44.455,A 0.015,B -0.000,C -180.000} C_DIS
LIN {X -399.692,Y 339.076,Z -44.467,A 0.015,B 0.000,C -180.000} C_DIS
LIN {X -400.552,Y 338.848,Z -44.498,A 0.015,B 0.000,C -180.000} C_DIS
LIN {X -400.596,Y 338.832,Z -44.500,A 0.015,B 0.000,C -180.000} C_DIS
LIN {X -400.134,Y 339.006,Z -44.500,A 0.015,B 0.000,C 180.000} C_DIS
LIN {X -398.924,Y 339.199,Z -44.500,A 0.015,B 0.000,C 180.000} C_DIS
LIN {X -213.380,Y 339.203,Z -44.500,A 0.015,B 0.000,C -180.000} C_DIS
LIN {X -213.561,Y 339.162,Z -44.500,A 0.015,B 0.000,C 180.000} C_DIS
LIN {X -214.650,Y 338.882,Z -44.500,A 0.015,B 0.000,C -180.000} C_DIS
LIN {X -215.281,Y 338.651,Z -44.500,A 0.015,B 0.000,C 180.000} C_DIS
LIN {X -226.164,Y 333.382,Z -44.500,A 0.015,B 0.000,C -180.000} C_DIS
LIN {X -226.674,Y 333.077,Z -44.500,A 0.015,B 0.000,C -180.000} C_DIS
LIN {X -228.125,Y 332.027,Z -44.500,A 0.015,B 0.000,C 180.000} C_DIS
LIN {X -228.464,Y 331.746,Z -44.500,A 0.015,B 0.000,C 180.000} C_DIS
LIN {X -236.648,Y 324.014,Z -44.500,A 0.015,B 0.000,C 180.000} C_DIS
LIN {X -236.966,Y 323.669,Z -44.500,A 0.015,B 0.000,C -180.000} C_DIS
LIN {X -237.837,Y 322.581,Z -44.500,A 0.015,B 0.000,C 180.000} C_DIS
LIN {X -238.117,Y 322.172,Z -44.500,A 0.015,B 0.000,C 180.000} C_DIS
LIN {X -240.445,Y 318.182,Z -44.500,A 0.015,B -0.000,C -180.000} C_DIS
LIN {X -240.483,Y 318.115,Z -44.500,A 0.015,B -0.000,C 180.000} C_DIS
LIN {X -243.694,Y 312.311,Z -44.500,A 0.015,B 0.000,C 180.000} C_DIS
LIN {X -243.876,Y 311.927,Z -44.500,A 0.015,B -0.000,C -180.000} C_DIS
LIN {X -244.744,Y 309.750,Z -44.500,A 0.015,B -0.000,C -180.000} C_DIS
LIN {X -244.946,Y 309.009,Z -44.500,A 0.015,B 0.000,C -180.000} C_DIS
LIN {X -246.389,Y 299.577,Z -44.500,A 0.015,B -0.000,C -180.000} C_DIS
LIN {X -246.415,Y 299.356,Z -44.500,A 0.015,B 0.000,C -180.000} C_DIS
LIN {X -246.509,Y 298.268,Z -44.500,A 0.015,B -0.000,C 180.000} C_DIS
CIRC {X -246.514,Y 297.752,Z -44.500,A 0.015,B 0.000,C -180.000},{X -246.441,Y 297.240,Z -44.500,A 0.015,B -0.000,C 180.000} C_DIS
LIN {X -245.042,Y 290.980,Z -44.500,A 0.015,B 0.000,C 180.000} C_DIS
LIN {X -245.027,Y 290.913,Z -44.500,A 0.015,B 0.000,C 180.000} C_DIS
LIN {X -244.073,Y 287.016,Z -44.500,A 0.015,B 0.000,C 180.000} C_DIS
LIN {X -243.737,Y 286.165,Z -44.500,A 0.015,B 0.000,C -180.000} C_DIS
LIN {X -241.012,Y 281.309,Z -44.500,A 0.015,B 0.000,C 180.000} C_DIS
LIN {X -240.643,Y 280.778,Z -44.500,A 0.015,B 0.000,C 180.000} C_DIS
LIN {X -237.074,Y 276.566,Z -44.500,A 0.015,B 0.000,C 180.000} C_DIS
LIN {X -236.515,Y 276.041,Z -44.500,A 0.015,B 0.000,C 180.000} C_DIS
LIN {X -230.703,Y 271.706,Z -44.500,A 0.015,B 0.000,C 180.000} C_DIS
LIN {X -230.157,Y 271.374,Z -44.500,A 0.015,B 0.000,C -180.000} C_DIS
LIN {X -227.128,Y 269.905,Z -44.500,A 0.015,B 0.000,C -180.000} C_DIS
LIN {X -226.735,Y 269.744,Z -44.500,A 0.015,B 0.000,C -180.000} C_DIS
LIN {X -222.871,Y 268.438,Z -44.500,A 0.015,B -0.000,C -180.000} C_DIS
LIN {X -222.224,Y 268.288,Z -44.500,A 0.015,B 0.000,C 180.000} C_DIS
LIN {X -215.331,Y 267.392,Z -44.500,A 0.015,B 0.000,C -180.000} C_DIS
LIN {X -214.895,Y 267.364,Z -44.500,A 0.015,B 0.000,C -180.000} C_DIS
LIN {X -178.617,Y 267.364,Z -44.500,A 0.015,B 0.000,C 180.000} C_DIS
LIN {X -178.181,Y 267.392,Z -44.500,A 0.015,B 0.000,C -180.000} C_DIS
LIN {X -171.288,Y 268.288,Z -44.500,A 0.015,B -0.000,C 180.000} C_DIS
LIN {X -170.681,Y 268.425,Z -44.500,A 0.015,B 0.000,C -180.000} C_DIS
LIN {X -167.479,Y 269.462,Z -44.500,A 0.015,B 0.000,C 180.000} C_DIS
LIN {X -167.082,Y 269.620,Z -44.500,A 0.015,B 0.000,C 180.000} C_DIS
LIN {X -163.390,Y 271.357,Z -44.500,A 0.015,B 0.000,C -180.000} C_DIS
LIN {X -162.809,Y 271.706,Z -44.500,A 0.015,B 0.000,C -180.000} C_DIS
LIN {X -156.996,Y 276.041,Z -44.500,A 0.015,B 0.000,C 180.000} C_DIS
LIN {X -156.438,Y 276.566,Z -44.500,A 0.015,B 0.000,C 180.000} C_DIS
LIN {X -152.869,Y 280.778,Z -44.500,A 0.015,B 0.000,C -180.000} C_DIS
LIN {X -152.500,Y 281.309,Z -44.500,A 0.015,B 0.000,C -180.000} C_DIS
LIN {X -149.775,Y 286.165,Z -44.500,A 0.015,B 0.000,C -180.000} C_DIS
LIN {X -149.433,Y 287.042,Z -44.500,A 0.015,B 0.000,C 180.000} C_DIS
LIN {X -147.115,Y 296.836,Z -44.500,A 0.015,B -0.000,C -180.000} C_DIS
LIN {X -147.028,Y 297.457,Z -44.500,A 0.015,B 0.000,C 180.000} C_DIS
LIN {X -146.994,Y 298.183,Z -44.500,A 0.015,B 0.000,C -180.000} C_DIS
LIN {X -147.027,Y 298.837,Z -44.500,A 0.015,B 0.000,C 180.000} C_DIS
LIN {X -148.481,Y 308.631,Z -44.500,A 0.015,B 0.000,C 180.000} C_DIS
LIN {X -148.629,Y 309.238,Z -44.500,A 0.015,B 0.000,C 180.000} C_DIS
LIN {X -149.256,Y 311.052,Z -44.500,A 0.015,B 0.000,C 180.000} C_DIS
LIN {X -149.452,Y 311.509,Z -44.500,A 0.015,B 0.000,C -180.000} C_DIS
LIN {X -151.339,Y 315.136,Z -44.500,A 0.015,B 0.000,C 180.000} C_DIS
LIN {X -151.403,Y 315.253,Z -44.500,A 0.015,B 0.000,C -180.000} C_DIS
LIN {X -155.132,Y 321.783,Z -44.500,A 0.015,B 0.000,C 180.000} C_DIS
LIN {X -155.390,Y 322.169,Z -44.500,A 0.015,B 0.000,C 180.000} C_DIS
LIN {X -156.507,Y 323.620,Z -44.500,A 0.015,B 0.000,C 180.000} C_DIS
LIN {X -156.864,Y 324.014,Z -44.500,A 0.015,B 0.000,C 180.000} C_DIS
LIN {X -165.047,Y 331.746,Z -44.500,A 0.015,B 0.000,C 180.000} C_DIS
LIN {X -165.387,Y 332.027,Z -44.500,A 0.015,B -0.000,C 180.000} C_DIS
LIN {X -166.838,Y 333.077,Z -44.500,A 0.015,B 0.000,C 180.000} C_DIS
LIN {X -167.341,Y 333.379,Z -44.500,A 0.015,B 0.000,C 180.000} C_DIS
LIN {X -177.862,Y 338.499,Z -44.500,A 0.015,B 0.000,C 180.000} C_DIS
LIN {X -178.267,Y 338.664,Z -44.500,A 0.015,B 0.000,C 180.000} C_DIS
LIN {X -179.356,Y 339.029,Z -44.500,A 0.015,B -0.000,C 180.000} C_DIS
LIN {X -179.925,Y 339.166,Z -44.500,A 0.015,B -0.000,C 180.000} C_DIS
LIN {X -180.175,Y 339.204,Z -44.500,A 0.015,B 0.000,C -180.000} C_DIS
LIN {X 4.865,Y 339.209,Z -44.500,A 0.015,B 0.000,C 180.000} C_DIS
LIN {X 5.937,Y 339.152,Z -44.500,A 0.015,B 0.000,C -180.000} C_DIS
LIN {X 6.802,Y 338.955,Z -44.500,A 0.015,B -0.000,C 180.000} C_DIS
LIN {X 7.069,Y 338.840,Z -44.500,A 0.015,B 0.000,C -180.000} C_DIS
LIN {X 7.566,Y 338.456,Z -44.330,A 0.015,B 0.000,C -180.000} C_DIS
LIN {X 7.779,Y 338.046,Z -43.865,A 0.015,B -0.000,C 180.000} C_DIS
LIN {X 7.818,Y 337.880,Z -43.230,A 0.015,B 0.000,C -180.000} C_DIS
$VEL.CP = 1.00000
LIN {X 7.818,Y 337.880,Z 11.000,A 0.015,B -0.000,C 180.000} C_DIS
$VEL.CP = 1.00000
LIN {X 10.265,Y 334.347,Z 11.000,A 0.015,B -0.000,C -180.000} C_DIS
$VEL.CP = 0.10000
LIN {X 10.265,Y 334.347,Z -29.000,A 0.015,B 0.000,C 180.000} C_DIS
LIN {X 10.265,Y 334.347,Z -44.500,A 0.015,B 0.000,C 180.000} C_DIS
LIN {X 10.273,Y 31.933,Z -44.500,A 0.015,B 0.000,C -180.000} C_DIS
LIN {X 9.285,Y 36.109,Z -44.500,A 0.015,B -0.000,C -180.000} C_DIS
LIN {X 9.155,Y 36.530,Z -44.500,A 0.015,B -0.000,C 180.000} C_DIS
LIN {X 8.502,Y 38.250,Z -44.500,A 0.015,B 0.000,C -180.000} C_DIS
LIN {X 8.269,Y 38.741,Z -44.500,A 0.015,B 0.000,C -180.000} C_DIS
LIN {X 6.110,Y 42.480,Z -44.500,A 0.015,B 0.000,C -180.000} C_DIS
LIN {X 6.079,Y 42.533,Z -44.500,A 0.015,B -0.000,C -180.000} C_DIS
LIN {X 2.586,Y 48.337,Z -44.500,A 0.015,B 0.000,C -180.000} C_DIS
LIN {X 2.352,Y 48.677,Z -44.500,A 0.015,B -0.000,C 180.000} C_DIS
LIN {X 1.028,Y 50.369,Z -44.500,A 0.015,B 0.000,C -180.000} C_DIS
LIN {X 0.484,Y 50.921,Z -44.500,A 0.015,B 0.000,C -180.000} C_DIS
LIN {X -7.437,Y 57.295,Z -44.500,A 0.015,B 0.000,C -180.000} C_DIS
LIN {X -7.808,Y 57.555,Z -44.500,A 0.015,B 0.000,C 180.000} C_DIS
LIN {X -8.472,Y 57.956,Z -44.500,A 0.015,B 0.000,C 180.000} C_DIS
LIN {X -9.243,Y 58.298,Z -44.500,A 0.015,B -0.000,C -180.000} C_DIS
LIN {X -19.100,Y 61.276,Z -44.500,A 0.015,B 0.000,C -180.000} C_DIS
LIN {X -20.032,Y 61.420,Z -44.500,A 0.015,B 0.000,C 180.000} C_DIS
LIN {X -25.473,Y 61.495,Z -44.500,A 0.015,B 0.000,C 180.000} C_DIS
LIN {X -26.114,Y 61.442,Z -44.500,A 0.015,B 0.000,C -180.000} C_DIS
LIN {X -31.556,Y 60.471,Z -44.500,A 0.015,B -0.000,C 180.000} C_DIS
LIN {X -32.284,Y 60.255,Z -44.500,A 0.015,B 0.000,C -180.000} C_DIS
LIN {X -38.814,Y 57.482,Z -44.500,A 0.015,B 0.000,C 180.000} C_DIS
LIN {X -39.365,Y 57.185,Z -44.500,A 0.015,B 0.000,C 180.000} C_DIS
LIN {X -42.330,Y 55.213,Z -44.500,A 0.015,B -0.000,C -180.000} C_DIS
LIN {X -42.678,Y 54.948,Z -44.500,A 0.015,B 0.000,C -180.000} C_DIS
LIN {X -45.688,Y 52.326,Z -44.500,A 0.015,B 0.000,C 180.000} C_DIS
LIN {X -46.147,Y 51.839,Z -44.500,A 0.015,B 0.000,C 180.000} C_DIS
LIN {X -50.396,Y 46.321,Z -44.500,A 0.015,B 0.000,C 180.000} C_DIS
LIN {X -50.645,Y 45.950,Z -44.500,A 0.015,B 0.000,C -180.000} C_DIS
LIN {X -68.791,Y 14.550,Z -44.500,A 0.015,B 0.000,C 180.000} C_DIS
LIN {X -68.983,Y 14.163,Z -44.500,A 0.015,B 0.000,C 180.000} C_DIS
LIN {X -71.720,Y 7.619,Z -44.500,A 0.015,B -0.000,C -180.000} C_DIS
LIN {X -71.908,Y 7.020,Z -44.500,A 0.015,B 0.000,C 180.000} C_DIS
LIN {X -72.602,Y 3.770,Z -44.500,A 0.015,B 0.000,C 180.000} C_DIS
LIN {X -72.663,Y 3.360,Z -44.500,A 0.015,B 0.000,C -180.000} C_DIS
LIN {X -73.014,Y -0.630,Z -44.500,A 0.015,B 0.000,C 180.000} C_DIS
LIN {X -73.005,Y -1.312,Z -44.500,A 0.015,B -0.000,C 180.000} C_DIS
LIN {X -72.173,Y -8.567,Z -44.500,A 0.015,B 0.000,C -180.000} C_DIS
LIN {X -72.004,Y -9.303,Z -44.500,A 0.015,B 0.000,C -180.000} C_DIS
LIN {X -70.782,Y -12.780,Z -44.500,A 0.015,B 0.000,C 180.000} C_DIS
LIN {X -70.164,Y -14.482,Z -44.500,A 0.015,B 0.000,C 180.000} C_DIS
LIN {X -69.916,Y -15.015,Z -44.500,A 0.015,B 0.000,C 180.000} C_DIS
LIN {X -67.656,Y -18.938,Z -44.500,A 0.015,B 0.000,C 180.000} C_DIS
LIN {X -67.535,Y -19.133,Z -44.500,A 0.015,B -0.000,C 180.000} C_DIS
LIN {X -66.788,Y -20.248,Z -44.500,A 0.015,B 0.000,C 180.000} C_DIS
LIN {X -66.297,Y -20.828,Z -44.500,A 0.015,B 0.000,C -180.000} C_DIS
LIN {X -59.763,Y -26.977,Z -44.500,A 0.015,B 0.000,C -180.000} C_DIS
LIN {X -59.602,Y -27.119,Z -44.500,A 0.015,B 0.000,C 180.000} C_DIS
LIN {X -58.514,Y -28.020,Z -44.500,A 0.015,B -0.000,C -180.000} C_DIS
CIRC {X -58.082,Y -28.324,Z -44.500,A 0.015,B 0.000,C 180.000},{X -57.609,Y -28.557,Z -44.500,A 0.015,B 0.000,C -180.000} C_DIS
LIN {X -50.808,Y -31.266,Z -44.500,A 0.015,B 0.000,C 180.000} C_DIS
LIN {X -342.732,Y -31.266,Z -44.500,A 0.015,B -0.000,C 180.000} C_DIS
LIN {X -336.289,Y -28.753,Z -44.500,A 0.015,B 0.000,C 180.000} C_DIS
LIN {X -335.788,Y -28.508,Z -44.500,A 0.015,B 0.000,C 180.000} C_DIS
LIN {X -335.062,Y -28.076,Z -44.500,A 0.015,B -0.000,C -180.000} C_DIS
LIN {X -334.484,Y -27.642,Z -44.500,A 0.015,B -0.000,C 180.000} C_DIS
LIN {X -327.578,Y -21.194,Z -44.500,A 0.015,B 0.000,C -180.000} C_DIS
LIN {X -327.345,Y -20.954,Z -44.500,A 0.015,B 0.000,C -180.000} C_DIS
LIN {X -326.717,Y -20.239,Z -44.500,A 0.015,B -0.000,C -180.000} C_DIS
LIN {X -326.349,Y -19.732,Z -44.500,A 0.015,B 0.000,C 180.000} C_DIS
LIN {X -323.777,Y -15.392,Z -44.500,A 0.015,B -0.000,C 180.000} C_DIS
LIN {X -323.506,Y -14.820,Z -44.500,A 0.015,B -0.000,C -180.000} C_DIS
LIN {X -321.519,Y -9.334,Z -44.500,A 0.015,B -0.000,C -180.000} C_DIS
LIN {X -321.340,Y -8.581,Z -44.500,A 0.015,B -0.000,C -180.000} C_DIS
LIN {X -320.521,Y -1.689,Z -44.500,A 0.015,B -0.000,C 180.000} C_DIS
LIN {X -320.504,Y -1.073,Z -44.500,A 0.015,B 0.000,C 180.000} C_DIS
LIN {X -320.737,Y 2.554,Z -44.500,A 0.015,B -0.000,C -180.000} C_DIS
LIN {X -320.796,Y 3.005,Z -44.500,A 0.015,B 0.000,C -180.000} C_DIS
LIN {X -321.596,Y 6.981,Z -44.500,A 0.015,B 0.000,C 180.000} C_DIS
LIN {X -321.787,Y 7.609,Z -44.500,A 0.015,B 0.000,C 180.000} C_DIS
LIN {X -324.350,Y 13.790,Z -44.500,A 0.015,B 0.000,C -180.000} C_DIS
LIN {X -324.544,Y 14.184,Z -44.500,A 0.015,B 0.000,C 180.000} C_DIS
LIN {X -342.684,Y 45.663,Z -44.500,A 0.015,B 0.000,C -180.000} C_DIS
LIN {X -342.917,Y 46.015,Z -44.500,A 0.015,B -0.000,C 180.000} C_DIS
LIN {X -347.093,Y 51.536,Z -44.500,A 0.015,B 0.000,C -180.000} C_DIS
LIN {X -347.507,Y 51.991,Z -44.500,A 0.015,B 0.000,C 180.000} C_DIS
LIN {X -350.259,Y 54.508,Z -44.500,A 0.015,B -0.000,C -180.000} C_DIS
LIN {X -350.614,Y 54.791,Z -44.500,A 0.015,B -0.000,C -180.000} C_DIS
LIN {X -353.729,Y 56.953,Z -44.500,A 0.015,B 0.000,C -180.000} C_DIS
LIN {X -354.298,Y 57.272,Z -44.500,A 0.015,B 0.000,C -180.000} C_DIS
LIN {X -360.828,Y 60.138,Z -44.500,A 0.015,B 0.000,C 180.000} C_DIS
LIN {X -361.573,Y 60.366,Z -44.500,A 0.015,B -0.000,C -180.000} C_DIS
LIN {X -367.378,Y 61.439,Z -44.500,A 0.015,B 0.000,C 180.000} C_DIS
LIN {X -368.038,Y 61.495,Z -44.500,A 0.015,B -0.000,C 180.000} C_DIS
LIN {X -373.480,Y 61.420,Z -44.500,A 0.015,B 0.000,C -180.000} C_DIS
LIN {X -374.400,Y 61.280,Z -44.500,A 0.015,B 0.000,C -180.000} C_DIS
LIN {X -383.593,Y 58.540,Z -44.500,A 0.015,B 0.000,C -180.000} C_DIS
LIN {X -383.927,Y 58.422,Z -44.500,A 0.015,B 0.000,C -180.000} C_DIS
LIN {X -384.922,Y 58.008,Z -44.500,A 0.015,B -0.000,C 180.000} C_DIS
LIN {X -385.722,Y 57.537,Z -44.500,A 0.015,B 0.000,C 180.000} C_DIS
LIN {X -393.652,Y 51.259,Z -44.500,A 0.015,B 0.000,C 180.000} C_DIS
LIN {X -394.131,Y 50.797,Z -44.500,A 0.015,B 0.000,C -180.000} C_DIS
LIN {X -395.533,Y 49.145,Z -44.500,A 0.015,B 0.000,C 180.000} C_DIS
LIN {X -395.823,Y 48.748,Z -44.500,A 0.015,B -0.000,C -180.000} C_DIS
LIN {X -397.862,Y 45.482,Z -44.500,A 0.015,B -0.000,C -180.000} C_DIS
LIN {X -397.917,Y 45.390,Z -44.500,A 0.015,B 0.000,C -180.000} C_DIS
LIN {X -401.777,Y 38.749,Z -44.500,A 0.015,B -0.000,C -180.000} C_DIS
LIN {X -402.014,Y 38.250,Z -44.500,A 0.015,B 0.000,C 180.000} C_DIS
LIN {X -402.667,Y 36.530,Z -44.500,A 0.015,B -0.000,C 180.000} C_DIS
LIN {X -402.797,Y 36.109,Z -44.500,A 0.015,B -0.000,C 180.000} C_DIS
LIN {X -403.779,Y 31.961,Z -44.500,A 0.015,B 0.000,C -180.000} C_DIS
LIN {X -403.787,Y 333.800,Z -44.500,A 0.015,B -0.000,C -180.000} C_DIS
LIN {X -403.730,Y 334.871,Z -44.500,A 0.015,B -0.000,C -180.000} C_DIS
LIN {X -403.533,Y 335.736,Z -44.500,A 0.015,B 0.000,C -180.000} C_DIS
LIN {X -403.418,Y 336.003,Z -44.500,A 0.015,B 0.000,C 180.000} C_DIS
LIN {X -403.034,Y 336.500,Z -44.330,A 0.015,B -0.000,C 180.000} C_DIS
LIN {X -402.624,Y 336.714,Z -43.865,A 0.015,B -0.000,C -180.000} C_DIS
LIN {X -402.458,Y 336.753,Z -43.230,A 0.015,B 0.000,C -180.000} C_DIS
$VEL.CP = 1.00000
LIN {X -402.458,Y 336.753,Z 11.000,A 0.015,B 0.000,C 180.000} C_DIS
$VEL.CP = 1.00000
LIN {X -328.209,Y 254.069,Z 11.000,A 0.015,B 0.000,C 180.000} C_DIS
$VEL.CP = 1.00000
LIN {X -328.209,Y 254.069,Z -32.731,A 0.015,B 0.000,C -180.000} C_DIS
$VEL.CP = 0.10000
LIN {X -328.047,Y 254.050,Z -33.353,A 0.015,B 0.000,C -180.000} C_DIS
LIN {X -327.601,Y 254.022,Z -33.816,A 0.015,B 0.000,C 180.000} C_DIS
LIN {X -326.986,Y 254.037,Z -34.000,A 0.015,B 0.000,C -180.000} C_DIS
LIN {X -321.749,Y 258.062,Z -34.244,A 0.015,B 0.000,C -180.000} C_DIS
LIN {X -323.338,Y 264.472,Z -34.488,A 0.015,B 0.000,C -180.000} C_DIS
LIN {X -329.848,Y 265.585,Z -34.732,A 0.015,B 0.000,C 180.000} C_DIS
LIN {X -333.476,Y 260.067,Z -34.976,A 0.015,B -0.000,C 180.000} C_DIS
LIN {X -329.874,Y 254.531,Z -35.220,A 0.015,B -0.000,C 180.000} C_DIS
LIN {X -323.359,Y 255.613,Z -35.464,A 0.015,B -0.000,C 180.000} C_DIS
LIN {X -321.740,Y 262.016,Z -35.708,A 0.015,B -0.000,C 180.000} C_DIS
LIN {X -326.956,Y 266.065,Z -35.952,A 0.015,B 0.000,C 180.000} C_DIS
LIN {X -332.757,Y 262.908,Z -36.196,A 0.015,B 0.000,C -180.000} C_DIS
LIN {X -332.189,Y 256.329,Z -36.440,A 0.015,B 0.000,C -180.000} C_DIS
LIN {X -325.933,Y 254.212,Z -36.685,A 0.015,B 0.000,C 180.000} C_DIS
LIN {X -321.488,Y 259.096,Z -36.929,A 0.015,B 0.000,C -180.000} C_DIS
LIN {X -324.180,Y 265.126,Z -37.173,A 0.015,B 0.000,C -180.000} C_DIS
LIN {X -330.784,Y 265.075,Z -37.417,A 0.015,B 0.000,C -180.000} C_DIS
LIN {X -333.384,Y 259.004,Z -37.661,A 0.015,B 0.000,C -180.000} C_DIS
LIN {X -328.864,Y 254.190,Z -37.905,A 0.015,B 0.000,C -180.000} C_DIS
LIN {X -322.641,Y 256.402,Z -38.149,A 0.015,B -0.000,C 180.000} C_DIS
LIN {X -322.174,Y 262.990,Z -38.393,A 0.015,B 0.000,C 180.000} C_DIS
LIN {X -328.023,Y 266.057,Z -38.637,A 0.015,B 0.000,C 180.000} C_DIS
LIN {X -333.177,Y 261.928,Z -38.881,A 0.015,B 0.000,C 180.000} C_DIS
LIN {X -331.459,Y 255.551,Z -39.125,A 0.015,B 0.000,C -180.000} C_DIS
LIN {X -324.928,Y 254.569,Z -39.369,A 0.015,B 0.000,C -180.000} C_DIS
LIN {X -321.412,Y 260.160,Z -39.613,A 0.015,B 0.000,C 180.000} C_DIS
LIN {X -325.125,Y 265.622,Z -39.857,A 0.015,B 0.000,C 180.000} C_DIS
LIN {X -331.617,Y 264.409,Z -40.101,A 0.015,B 0.000,C 180.000} C_DIS
LIN {X -333.107,Y 257.975,Z -40.345,A 0.015,B 0.000,C 180.000} C_DIS
LIN {X -327.809,Y 254.031,Z -40.589,A 0.015,B -0.000,C -180.000} C_DIS
LIN {X -322.073,Y 257.305,Z -40.833,A 0.015,B 0.000,C -180.000} C_DIS
LIN {X -322.774,Y 263.872,Z -41.077,A 0.015,B -0.000,C 180.000} C_DIS
LIN {X -329.072,Y 265.861,Z -41.321,A 0.015,B 0.000,C 180.000} C_DIS
LIN {X -333.418,Y 260.889,Z -41.565,A 0.015,B 0.000,C 180.000} C_DIS
LIN {X -330.604,Y 254.914,Z -41.810,A 0.015,B 0.000,C 180.000} C_DIS
LIN {X -324.002,Y 255.098,Z -42.054,A 0.015,B 0.000,C -180.000} C_DIS
LIN {X -321.525,Y 261.220,Z -42.298,A 0.015,B 0.000,C -180.000} C_DIS
LIN {X -326.142,Y 265.943,Z -42.542,A 0.015,B 0.000,C 180.000} C_DIS
LIN {X -332.319,Y 263.605,Z -42.786,A 0.015,B 0.000,C 180.000} C_DIS
LIN {X -332.652,Y 257.010,Z -43.030,A 0.015,B 0.000,C 180.000} C_DIS
LIN {X -326.743,Y 254.061,Z -43.274,A 0.015,B 0.000,C 180.000} C_DIS
LIN {X -321.673,Y 258.293,Z -43.518,A 0.015,B 0.000,C 180.000} C_DIS
LIN {X -323.520,Y 264.634,Z -43.762,A 0.015,B 0.000,C 180.000} C_DIS
LIN {X -330.069,Y 265.484,Z -44.006,A 0.015,B 0.000,C 180.000} C_DIS
LIN {X -333.472,Y 259.823,Z -44.250,A 0.015,B -0.000,C 180.000} C_DIS
LIN {X -329.649,Y 254.438,Z -44.494,A 0.015,B 0.000,C -180.000} C_DIS
LIN {X -323.183,Y 255.782,Z -44.738,A 0.015,B 0.000,C 180.000} C_DIS
LIN {X -321.824,Y 262.245,Z -44.982,A 0.015,B 0.000,C 180.000} C_DIS
LIN {X -327.200,Y 266.080,Z -45.226,A 0.015,B 0.000,C 180.000} C_DIS
LIN {X -332.868,Y 262.691,Z -45.470,A 0.015,B -0.000,C 180.000} C_DIS
LIN {X -332.035,Y 256.140,Z -45.714,A 0.015,B 0.000,C 180.000} C_DIS
LIN {X -325.699,Y 254.278,Z -45.958,A 0.015,B 0.000,C -180.000} C_DIS
LIN {X -321.454,Y 259.337,Z -46.202,A 0.015,B 0.000,C 180.000} C_DIS
LIN {X -324.388,Y 265.254,Z -46.446,A 0.015,B 0.000,C 180.000} C_DIS
LIN {X -330.985,Y 264.936,Z -46.690,A 0.015,B 0.000,C 180.000} C_DIS
LIN {X -333.337,Y 258.765,Z -46.935,A 0.015,B 0.000,C 180.000} C_DIS
LIN {X -328.626,Y 254.137,Z -47.179,A 0.015,B 0.000,C 180.000} C_DIS
LIN {X -322.498,Y 256.599,Z -47.423,A 0.015,B 0.000,C -180.000} C_DIS
LIN {X -322.297,Y 263.200,Z -47.667,A 0.015,B 0.000,C 180.000} C_DIS
LIN {X -328.265,Y 266.029,Z -47.911,A 0.015,B 0.000,C 180.000} C_DIS
LIN {X -333.248,Y 261.694,Z -48.155,A 0.015,B 0.000,C -180.000} C_DIS
LIN {X -331.274,Y 255.392,Z -48.399,A 0.015,B -0.000,C 180.000} C_DIS
LIN {X -324.709,Y 254.676,Z -48.643,A 0.015,B 0.000,C 180.000} C_DIS
LIN {X -321.421,Y 260.404,Z -48.887,A 0.015,B 0.000,C 180.000} C_DIS
LIN {X -325.352,Y 265.711,Z -49.131,A 0.015,B -0.000,C 180.000} C_DIS
LIN {X -331.790,Y 264.236,Z -49.375,A 0.015,B 0.000,C -180.000} C_DIS
LIN {X -333.018,Y 257.747,Z -49.619,A 0.015,B -0.000,C -180.000} C_DIS
LIN {X -327.565,Y 254.021,Z -49.863,A 0.015,B 0.000,C -180.000} C_DIS
LIN {X -321.967,Y 257.524,Z -50.107,A 0.015,B 0.000,C -180.000} C_DIS
LIN {X -322.932,Y 264.057,Z -50.351,A 0.015,B 0.000,C 180.000} C_DIS
LIN {X -329.305,Y 265.791,Z -50.595,A 0.015,B 0.000,C -180.000} C_DIS
LIN {X -333.447,Y 260.646,Z -50.839,A 0.015,B 0.000,C 180.000} C_DIS
LIN {X -330.393,Y 254.790,Z -51.083,A 0.015,B 0.000,C 180.000} C_DIS
LIN {X -323.805,Y 255.241,Z -51.327,A 0.015,B 0.000,C 180.000} C_DIS
LIN {X -321.577,Y 261.459,Z -51.571,A 0.015,B -0.000,C 180.000} C_DIS
LIN {X -326.381,Y 265.991,Z -51.815,A 0.015,B 0.000,C 180.000} C_DIS
LIN {X -332.459,Y 263.405,Z -52.060,A 0.015,B 0.000,C 180.000} C_DIS
LIN {X -332.525,Y 256.801,Z -52.304,A 0.015,B -0.000,C 180.000} C_DIS
LIN {X -326.501,Y 254.094,Z -52.548,A 0.015,B 0.000,C 180.000} C_DIS
LIN {X -321.607,Y 258.528,Z -52.792,A 0.015,B -0.000,C 180.000} C_DIS
LIN {X -323.708,Y 264.789,Z -53.036,A 0.015,B 0.000,C -180.000} C_DIS
LIN {X -330.287,Y 265.373,Z -53.280,A 0.015,B -0.000,C 180.000} C_DIS
LIN {X -333.458,Y 259.580,Z -53.524,A 0.015,B 0.000,C 180.000} C_DIS
LIN {X -329.420,Y 254.353,Z -53.768,A 0.015,B -0.000,C 180.000} C_DIS
LIN {X -323.014,Y 255.957,Z -54.012,A 0.015,B 0.000,C -180.000} C_DIS
LIN {X -321.917,Y 262.470,Z -54.256,A 0.015,B -0.000,C 180.000} C_DIS
LIN {X -327.444,Y 266.085,Z -54.500,A 0.015,B 0.000,C 180.000} C_DIS
LIN {X -327.831,Y 266.085,Z -54.500,A 0.015,B 0.000,C 180.000} C_DIS
CIRC {X -329.838,Y 265.254,Z -54.500,A 0.015,B -0.000,C -180.000},{X -330.669,Y 263.246,Z -54.500,A 0.015,B -0.000,C 180.000} C_DIS
LIN {X -330.668,Y 221.143,Z -54.500,A 0.015,B 0.000,C 180.000} C_DIS
CIRC {X -329.579,Y 219.999,Z -54.500,A 0.015,B -0.000,C -180.000},{X -328.382,Y 221.029,Z -54.500,A 0.015,B 0.000,C 180.000} C_DIS
LIN {X -324.192,Y 262.964,Z -54.500,A 0.015,B -0.000,C -180.000} C_DIS
CIRC {X -324.912,Y 265.151,Z -54.500,A 0.015,B 0.000,C -180.000},{X -327.016,Y 266.085,Z -54.500,A 0.015,B 0.000,C 180.000} C_DIS
LIN {X -327.444,Y 266.085,Z -54.500,A 0.015,B 0.000,C 180.000} C_DIS
CIRC {X -329.629,Y 266.879,Z -54.500,A 0.015,B -0.000,C -180.000},{X -330.794,Y 268.892,Z -54.500,A 0.015,B -0.000,C 180.000} C_DIS
CIRC {X -332.529,Y 270.803,Z -54.500,A 0.015,B 0.000,C -180.000},{X -335.003,Y 270.069,Z -54.500,A 0.015,B -0.000,C 180.000} C_DIS
CIRC {X -335.715,Y 268.884,Z -54.500,A 0.015,B 0.000,C 180.000},{X -335.962,Y 267.525,Z -54.500,A 0.015,B 0.000,C -180.000} C_DIS
LIN {X -335.960,Y 181.590,Z -54.500,A 0.015,B 0.000,C -180.000} C_DIS
CIRC {X -334.847,Y 179.767,Z -54.500,A 0.015,B -0.000,C 180.000},{X -332.717,Y 179.926,Z -54.500,A 0.015,B 0.000,C 180.000} C_DIS
LIN {X -328.137,Y 183.215,Z -54.500,A 0.015,B -0.000,C 180.000} C_DIS
CIRC {X -327.061,Y 184.403,Z -54.500,A 0.015,B 0.000,C -180.000},{X -326.570,Y 185.927,Z -54.500,A 0.015,B 0.000,C -180.000} C_DIS
LIN {X -318.408,Y 267.614,Z -54.500,A 0.015,B 0.000,C -180.000} C_DIS
CIRC {X -319.276,Y 270.252,Z -54.500,A 0.015,B -0.000,C 180.000},{X -321.815,Y 271.378,Z -54.500,A 0.015,B 0.000,C -180.000} C_DIS
LIN {X -332.110,Y 271.378,Z -54.500,A 0.015,B 0.000,C 180.000} C_DIS
CIRC {X -333.698,Y 271.035,Z -54.500,A 0.015,B 0.000,C -180.000},{X -335.003,Y 270.069,Z -54.500,A 0.015,B 0.000,C 180.000} C_DIS
CIRC {X -337.398,Y 267.896,Z -54.500,A 0.015,B 0.000,C 180.000},{X -340.218,Y 266.315,Z -54.500,A 0.015,B -0.000,C 180.000} C_DIS
CIRC {X -342.803,Y 264.176,Z -54.500,A 0.015,B 0.000,C -180.000},{X -343.773,Y 260.964,Z -54.500,A 0.015,B 0.000,C 180.000} C_DIS
LIN {X -343.770,Y 166.365,Z -54.500,A 0.015,B 0.000,C 180.000} C_DIS
CIRC {X -342.657,Y 164.542,Z -54.500,A 0.015,B -0.000,C 180.000},{X -340.527,Y 164.701,Z -54.500,A 0.015,B 0.000,C 180.000} C_DIS
LIN {X -323.779,Y 176.729,Z -54.500,A 0.015,B -0.000,C -180.000} C_DIS
CIRC {X -320.343,Y 180.522,Z -54.500,A 0.015,B 0.000,C -180.000},{X -318.774,Y 185.393,Z -54.500,A 0.015,B 0.000,C -180.000} C_DIS
LIN {X -309.777,Y 275.425,Z -54.500,A 0.015,B 0.000,C 180.000} C_DIS
CIRC {X -310.646,Y 278.063,Z -54.500,A 0.015,B 0.000,C 180.000},{X -313.184,Y 279.189,Z -54.500,A 0.015,B 0.000,C -180.000} C_DIS
LIN {X -339.921,Y 279.189,Z -54.500,A 0.015,B 0.000,C -180.000} C_DIS
CIRC {X -342.645,Y 278.060,Z -54.500,A 0.015,B -0.000,C 180.000},{X -343.773,Y 275.335,Z -54.500,A 0.015,B -0.000,C -180.000} C_DIS
LIN {X -343.773,Y 260.964,Z -54.500,A 0.015,B 0.000,C -180.000} C_DIS
CIRC {X -344.839,Y 257.443,Z -54.500,A 0.015,B 0.000,C 180.000},{X -347.678,Y 255.105,Z -54.500,A 0.015,B 0.000,C 180.000} C_DIS
CIRC {X -350.518,Y 252.768,Z -54.500,A 0.015,B -0.000,C -180.000},{X -351.584,Y 249.247,Z -54.500,A 0.015,B 0.000,C 180.000} C_DIS
LIN {X -351.581,Y 151.139,Z -54.500,A 0.015,B 0.000,C -180.000} C_DIS
CIRC {X -350.467,Y 149.317,Z -54.500,A 0.015,B 0.000,C 180.000},{X -348.338,Y 149.476,Z -54.500,A 0.015,B 0.000,C -180.000} C_DIS
LIN {X -316.620,Y 172.253,Z -54.500,A 0.015,B 0.000,C -180.000} C_DIS
CIRC {X -312.982,Y 176.270,Z -54.500,A 0.015,B 0.000,C -180.000},{X -311.320,Y 181.428,Z -54.500,A 0.015,B 0.000,C 180.000} C_DIS
LIN {X -301.147,Y 283.236,Z -54.500,A 0.015,B 0.000,C -180.000} C_DIS
CIRC {X -302.016,Y 285.874,Z -54.500,A 0.015,B 0.000,C -180.000},{X -304.554,Y 287.000,Z -54.500,A 0.015,B -0.000,C -180.000} C_DIS
LIN {X -347.732,Y 286.999,Z -54.500,A 0.015,B -0.000,C -180.000} C_DIS
CIRC {X -350.456,Y 285.871,Z -54.500,A 0.015,B 0.000,C 180.000},{X -351.584,Y 283.146,Z -54.500,A 0.015,B 0.000,C -180.000} C_DIS
LIN {X -351.584,Y 249.247,Z -54.500,A 0.015,B 0.000,C -180.000} C_DIS
CIRC {X -352.649,Y 245.727,Z -54.500,A 0.015,B -0.000,C 180.000},{X -355.489,Y 243.389,Z -54.500,A 0.015,B -0.000,C -180.000} C_DIS
CIRC {X -358.328,Y 241.051,Z -54.500,A 0.015,B 0.000,C -180.000},{X -359.394,Y 237.531,Z -54.500,A 0.015,B 0.000,C -180.000} C_DIS
LIN {X -359.391,Y 135.914,Z -54.500,A 0.015,B 0.000,C 180.000} C_DIS
CIRC {X -358.278,Y 134.092,Z -54.500,A 0.015,B -0.000,C -180.000},{X -356.148,Y 134.250,Z -54.500,A 0.015,B -0.000,C 180.000} C_DIS
LIN {X -309.198,Y 167.967,Z -54.500,A 0.015,B 0.000,C 180.000} C_DIS
CIRC {X -305.561,Y 171.984,Z -54.500,A 0.015,B 0.000,C -180.000},{X -303.899,Y 177.142,Z -54.500,A 0.015,B 0.000,C -180.000} C_DIS
LIN {X -292.517,Y 291.047,Z -54.500,A 0.015,B 0.000,C -180.000} C_DIS
CIRC {X -293.385,Y 293.685,Z -54.500,A 0.015,B 0.000,C 180.000},{X -295.924,Y 294.811,Z -54.500,A 0.015,B -0.000,C 180.000} C_DIS
LIN {X -355.543,Y 294.810,Z -54.500,A 0.015,B 0.000,C 180.000} C_DIS
CIRC {X -358.267,Y 293.681,Z -54.500,A 0.015,B -0.000,C 180.000},{X -359.396,Y 290.957,Z -54.500,A 0.015,B 0.000,C -180.000} C_DIS
LIN {X -359.394,Y 237.531,Z -54.500,A 0.015,B 0.000,C -180.000} C_DIS
CIRC {X -360.460,Y 234.010,Z -54.500,A 0.015,B -0.000,C 180.000},{X -363.299,Y 231.673,Z -54.500,A 0.015,B 0.000,C -180.000} C_DIS
CIRC {X -366.139,Y 229.335,Z -54.500,A 0.015,B -0.000,C -180.000},{X -367.205,Y 225.814,Z -54.500,A 0.015,B 0.000,C 180.000} C_DIS
LIN {X -367.202,Y 120.689,Z -54.500,A 0.015,B 0.000,C 180.000} C_DIS
CIRC {X -366.088,Y 118.867,Z -54.500,A 0.015,B 0.000,C 180.000},{X -363.958,Y 119.025,Z -54.500,A 0.015,B 0.000,C 180.000} C_DIS
LIN {X -301.777,Y 163.680,Z -54.500,A 0.015,B -0.000,C 180.000} C_DIS
CIRC {X -298.139,Y 167.697,Z -54.500,A 0.015,B 0.000,C -180.000},{X -296.477,Y 172.855,Z -54.500,A 0.015,B 0.000,C -180.000} C_DIS
LIN {X -283.887,Y 298.858,Z -54.500,A 0.015,B -0.000,C -180.000} C_DIS
CIRC {X -284.755,Y 301.496,Z -54.500,A 0.015,B -0.000,C -180.000},{X -287.294,Y 302.622,Z -54.500,A 0.015,B -0.000,C 180.000} C_DIS
LIN {X -363.354,Y 302.620,Z -54.500,A 0.015,B 0.000,C 180.000} C_DIS
CIRC {X -366.078,Y 301.492,Z -54.500,A 0.015,B -0.000,C -180.000},{X -367.207,Y 298.767,Z -54.500,A 0.015,B 0.000,C 180.000} C_DIS
LIN {X -367.205,Y 225.814,Z -54.500,A 0.015,B 0.000,C 180.000} C_DIS
CIRC {X -368.270,Y 222.294,Z -54.500,A 0.015,B 0.000,C -180.000},{X -371.110,Y 219.956,Z -54.500,A 0.015,B 0.000,C 180.000} C_DIS
CIRC {X -373.949,Y 217.618,Z -54.500,A 0.015,B 0.000,C -180.000},{X -375.015,Y 214.098,Z -54.500,A 0.015,B 0.000,C 180.000} C_DIS
LIN {X -375.012,Y 105.464,Z -54.500,A 0.015,B 0.000,C 180.000} C_DIS
CIRC {X -373.899,Y 103.641,Z -54.500,A 0.015,B -0.000,C 180.000},{X -371.769,Y 103.800,Z -54.500,A 0.015,B 0.000,C -180.000} C_DIS
LIN {X -293.711,Y 159.857,Z -54.500,A 0.015,B 0.000,C 180.000} C_DIS
CIRC {X -290.570,Y 163.325,Z -54.500,A 0.015,B 0.000,C 180.000},{X -289.135,Y 167.778,Z -54.500,A 0.015,B -0.000,C -180.000} C_DIS
LIN {X -275.474,Y 304.472,Z -54.500,A 0.015,B 0.000,C 180.000} C_DIS
CIRC {X -275.365,Y 305.060,Z -54.500,A 0.015,B -0.000,C 180.000},{X -275.237,Y 305.645,Z -54.500,A 0.015,B 0.000,C -180.000} C_DIS
CIRC {X -275.109,Y 306.229,Z -54.500,A 0.015,B 0.000,C 180.000},{X -274.999,Y 306.817,Z -54.500,A 0.015,B 0.000,C 180.000} C_DIS
CIRC {X -275.686,Y 309.334,Z -54.500,A 0.015,B 0.000,C 180.000},{X -278.052,Y 310.433,Z -54.500,A 0.015,B -0.000,C 180.000} C_DIS
LIN {X -371.165,Y 310.431,Z -54.500,A 0.015,B -0.000,C 180.000} C_DIS
CIRC {X -373.889,Y 309.302,Z -54.500,A 0.015,B 0.000,C 180.000},{X -375.018,Y 306.578,Z -54.500,A 0.015,B 0.000,C 180.000} C_DIS
LIN {X -375.015,Y 214.098,Z -54.500,A 0.015,B 0.000,C 180.000} C_DIS
CIRC {X -376.081,Y 210.578,Z -54.500,A 0.015,B 0.000,C 180.000},{X -378.920,Y 208.240,Z -54.500,A 0.015,B -0.000,C 180.000} C_DIS
CIRC {X -381.760,Y 205.902,Z -54.500,A 0.015,B 0.000,C -180.000},{X -382.826,Y 202.381,Z -54.500,A 0.015,B 0.000,C 180.000} C_DIS
LIN {X -382.822,Y 90.239,Z -54.500,A 0.015,B 0.000,C 180.000} C_DIS
CIRC {X -381.709,Y 88.416,Z -54.500,A 0.015,B 0.000,C -180.000},{X -379.579,Y 88.575,Z -54.500,A 0.015,B -0.000,C -180.000} C_DIS
LIN {X -287.927,Y 154.525,Z -54.500,A 0.015,B 0.000,C -180.000} C_DIS
CIRC {X -287.217,Y 154.999,Z -54.500,A 0.015,B 0.000,C -180.000},{X -286.479,Y 155.426,Z -54.500,A 0.015,B -0.000,C -180.000} C_DIS
CIRC {X -285.726,Y 155.826,Z -54.500,A 0.015,B 0.000,C 180.000},{X -284.971,Y 156.224,Z -54.500,A 0.015,B 0.000,C 180.000} C_DIS
CIRC {X -282.401,Y 158.704,Z -54.500,A 0.015,B 0.000,C 180.000},{X -281.571,Y 162.178,Z -54.500,A 0.015,B 0.000,C 180.000} C_DIS
CIRC {X -281.614,Y 163.091,Z -54.500,A 0.015,B 0.000,C 180.000},{X -281.651,Y 164.003,Z -54.500,A 0.015,B -0.000,C -180.000} C_DIS
CIRC {X -281.654,Y 164.917,Z -54.500,A 0.015,B 0.000,C -180.000},{X -281.594,Y 165.829,Z -54.500,A 0.015,B 0.000,C 180.000} C_DIS
LIN {X -267.483,Y 306.098,Z -54.500,A 0.015,B 0.000,C 180.000} C_DIS
CIRC {X -267.015,Y 308.301,Z -54.500,A 0.015,B 0.000,C -180.000},{X -266.369,Y 310.459,Z -54.500,A 0.015,B -0.000,C 180.000} C_DIS
CIRC {X -265.682,Y 312.602,Z -54.500,A 0.015,B 0.000,C -180.000},{X -265.088,Y 314.774,Z -54.500,A 0.015,B 0.000,C -180.000} C_DIS
CIRC {X -265.595,Y 317.170,Z -54.500,A 0.015,B 0.000,C -180.000},{X -267.797,Y 318.244,Z -54.500,A 0.015,B -0.000,C 180.000} C_DIS
LIN {X -378.976,Y 318.242,Z -54.500,A 0.015,B 0.000,C 180.000} C_DIS
CIRC {X -381.700,Y 317.113,Z -54.500,A 0.015,B 0.000,C 180.000},{X -382.829,Y 314.389,Z -54.500,A 0.015,B -0.000,C 180.000} C_DIS
LIN {X -382.825,Y 202.381,Z -54.500,A 0.015,B 0.000,C 180.000} C_DIS
CIRC {X -383.891,Y 198.861,Z -54.500,A 0.015,B 0.000,C 180.000},{X -386.731,Y 196.523,Z -54.500,A 0.015,B 0.000,C 180.000} C_DIS
CIRC {X -389.570,Y 194.185,Z -54.500,A 0.015,B -0.000,C 180.000},{X -390.636,Y 190.665,Z -54.500,A 0.015,B -0.000,C 180.000} C_DIS
LIN {X -390.633,Y 75.013,Z -54.500,A 0.015,B 0.000,C 180.000} C_DIS
CIRC {X -389.519,Y 73.191,Z -54.500,A 0.015,B -0.000,C 180.000},{X -387.390,Y 73.350,Z -54.500,A 0.015,B 0.000,C 180.000} C_DIS
LIN {X -283.475,Y 148.326,Z -54.500,A 0.015,B 0.000,C -180.000} C_DIS
CIRC {X -281.499,Y 149.534,Z -54.500,A 0.015,B 0.000,C 180.000},{X -279.366,Y 150.435,Z -54.500,A 0.015,B 0.000,C 180.000} C_DIS
CIRC {X -277.156,Y 151.108,Z -54.500,A 0.015,B -0.000,C 180.000},{X -274.909,Y 151.646,Z -54.500,A 0.015,B 0.000,C 180.000} C_DIS
CIRC {X -272.869,Y 153.107,Z -54.500,A 0.015,B 0.000,C 180.000},{X -272.579,Y 155.599,Z -54.500,A 0.015,B -0.000,C 180.000} C_DIS
CIRC {X -273.041,Y 157.191,Z -54.500,A 0.015,B 0.000,C 180.000},{X -273.442,Y 158.800,Z -54.500,A 0.015,B 0.000,C -180.000} C_DIS
CIRC {X -273.754,Y 160.429,Z -54.500,A 0.015,B 0.000,C 180.000},{X -273.945,Y 162.077,Z -54.500,A 0.015,B 0.000,C -180.000} C_DIS
CIRC {X -273.999,Y 162.824,Z -54.500,A 0.015,B 0.000,C -180.000},{X -274.043,Y 163.573,Z -54.500,A 0.015,B 0.000,C 180.000} C_DIS
CIRC {X -274.052,Y 164.322,Z -54.500,A 0.015,B 0.000,C 180.000},{X -274.006,Y 165.071,Z -54.500,A 0.015,B 0.000,C 180.000} C_DIS
LIN {X -259.860,Y 305.748,Z -54.500,A 0.015,B -0.000,C -180.000} C_DIS
CIRC {X -259.156,Y 308.544,Z -54.500,A 0.015,B 0.000,C -180.000},{X -258.323,Y 311.304,Z -54.500,A 0.015,B -0.000,C 180.000} C_DIS
CIRC {X -257.389,Y 314.031,Z -54.500,A 0.015,B 0.000,C -180.000},{X -256.382,Y 316.731,Z -54.500,A 0.015,B 0.000,C -180.000} C_DIS
CIRC {X -255.668,Y 318.300,Z -54.500,A 0.015,B -0.000,C -180.000},{X -254.781,Y 319.776,Z -54.500,A 0.015,B 0.000,C 180.000} C_DIS
CIRC {X -253.842,Y 321.218,Z -54.500,A 0.015,B 0.000,C -180.000},{X -252.964,Y 322.698,Z -54.500,A 0.015,B 0.000,C -180.000} C_DIS
CIRC {X -252.979,Y 324.939,Z -54.500,A 0.015,B -0.000,C -180.000},{X -254.923,Y 326.056,Z -54.500,A 0.015,B 0.000,C 180.000} C_DIS
LIN {X -386.787,Y 326.052,Z -54.500,A 0.015,B 0.000,C 180.000} C_DIS
CIRC {X -389.511,Y 324.924,Z -54.500,A 0.015,B 0.000,C -180.000},{X -390.640,Y 322.199,Z -54.500,A 0.015,B 0.000,C 180.000} C_DIS
LIN {X -390.636,Y 190.665,Z -54.500,A 0.015,B -0.000,C -180.000} C_DIS
LIN {X -390.481,Y 190.056,Z -54.330,A 0.015,B -0.000,C 180.000} C_DIS
LIN {X -390.189,Y 189.698,Z -53.865,A 0.015,B -0.000,C 180.000} C_DIS
LIN {X -390.052,Y 189.596,Z -53.230,A 0.015,B 0.000,C 180.000} C_DIS
$VEL.CP = 1.00000
LIN {X -390.052,Y 189.596,Z 11.000,A 0.015,B 0.000,C 180.000} C_DIS
$VEL.CP = 1.00000
LIN {X -206.449,Y 109.973,Z 11.000,A 0.015,B 0.000,C -180.000} C_DIS
$VEL.CP = 1.00000
LIN {X -206.449,Y 109.973,Z -32.731,A 0.015,B 0.000,C 180.000} C_DIS
$VEL.CP = 0.10000
LIN {X -206.467,Y 109.811,Z -33.353,A 0.015,B 0.000,C -180.000} C_DIS
LIN {X -206.495,Y 109.366,Z -33.816,A 0.015,B 0.000,C -180.000} C_DIS
LIN {X -206.480,Y 108.750,Z -34.000,A 0.015,B 0.000,C -180.000} C_DIS
LIN {X -202.456,Y 103.513,Z -34.244,A 0.015,B 0.000,C -180.000} C_DIS
LIN {X -196.045,Y 105.102,Z -34.488,A 0.015,B -0.000,C -180.000} C_DIS
LIN {X -194.932,Y 111.611,Z -34.732,A 0.015,B 0.000,C 180.000} C_DIS
LIN {X -200.450,Y 115.240,Z -34.976,A 0.015,B 0.000,C 180.000} C_DIS
LIN {X -205.986,Y 111.639,Z -35.220,A 0.015,B -0.000,C -180.000} C_DIS
LIN {X -204.905,Y 105.123,Z -35.464,A 0.015,B 0.000,C -180.000} C_DIS
LIN {X -198.502,Y 103.503,Z -35.708,A 0.015,B 0.000,C -180.000} C_DIS
LIN {X -194.452,Y 108.720,Z -35.952,A 0.015,B -0.000,C 180.000} C_DIS
LIN {X -197.609,Y 114.521,Z -36.196,A 0.015,B 0.000,C -180.000} C_DIS
LIN {X -204.189,Y 113.954,Z -36.440,A 0.015,B 0.000,C -180.000} C_DIS
LIN {X -206.305,Y 107.698,Z -36.685,A 0.015,B 0.000,C 180.000} C_DIS
LIN {X -201.422,Y 103.252,Z -36.929,A 0.015,B -0.000,C -180.000} C_DIS
LIN {X -195.391,Y 105.944,Z -37.173,A 0.015,B 0.000,C -180.000} C_DIS
LIN {X -195.442,Y 112.548,Z -37.417,A 0.015,B 0.000,C -180.000} C_DIS
LIN {X -201.513,Y 115.148,Z -37.661,A 0.015,B 0.000,C 180.000} C_DIS
LIN {X -206.328,Y 110.628,Z -37.905,A 0.015,B 0.000,C -180.000} C_DIS
LIN {X -204.116,Y 104.405,Z -38.149,A 0.015,B -0.000,C -180.000} C_DIS
LIN {X -197.528,Y 103.938,Z -38.393,A 0.015,B 0.000,C -180.000} C_DIS
LIN {X -194.460,Y 109.787,Z -38.637,A 0.015,B -0.000,C 180.000} C_DIS
LIN {X -198.589,Y 114.941,Z -38.881,A 0.015,B 0.000,C -180.000} C_DIS
LIN {X -204.966,Y 113.224,Z -39.125,A 0.015,B 0.000,C -180.000} C_DIS
LIN {X -205.948,Y 106.693,Z -39.369,A 0.015,B 0.000,C -180.000} C_DIS
LIN {X -200.358,Y 103.176,Z -39.613,A 0.015,B 0.000,C 180.000} C_DIS
LIN {X -194.896,Y 106.889,Z -39.857,A 0.015,B -0.000,C 180.000} C_DIS
LIN {X -196.109,Y 113.381,Z -40.101,A 0.015,B -0.000,C -180.000} C_DIS
LIN {X -202.543,Y 114.871,Z -40.345,A 0.015,B 0.000,C 180.000} C_DIS
LIN {X -206.486,Y 109.573,Z -40.589,A 0.015,B -0.000,C 180.000} C_DIS
LIN {X -203.213,Y 103.837,Z -40.833,A 0.015,B -0.000,C 180.000} C_DIS
LIN {X -196.646,Y 104.538,Z -41.077,A 0.015,B 0.000,C -180.000} C_DIS
LIN {X -194.656,Y 110.836,Z -41.321,A 0.015,B 0.000,C 180.000} C_DIS
LIN {X -199.629,Y 115.182,Z -41.565,A 0.015,B 0.000,C -180.000} C_DIS
LIN {X -205.603,Y 112.368,Z -41.810,A 0.015,B 0.000,C -180.000} C_DIS
LIN {X -205.419,Y 105.766,Z -42.054,A 0.015,B 0.000,C 180.000} C_DIS
LIN {X -199.297,Y 103.289,Z -42.298,A 0.015,B 0.000,C 180.000} C_DIS
LIN {X -194.575,Y 107.906,Z -42.542,A 0.015,B 0.000,C 180.000} C_DIS
LIN {X -196.912,Y 114.083,Z -42.786,A 0.015,B -0.000,C 180.000} C_DIS
LIN {X -203.508,Y 114.417,Z -43.030,A 0.015,B 0.000,C 180.000} C_DIS
LIN {X -206.457,Y 108.507,Z -43.274,A 0.015,B 0.000,C 180.000} C_DIS
LIN {X -202.224,Y 103.437,Z -43.518,A 0.015,B 0.000,C 180.000} C_DIS
LIN {X -195.883,Y 105.284,Z -43.762,A 0.015,B 0.000,C -180.000} C_DIS
LIN {X -195.034,Y 111.833,Z -44.006,A 0.015,B 0.000,C 180.000} C_DIS
LIN {X -200.694,Y 115.236,Z -44.250,A 0.015,B 0.000,C 180.000} C_DIS
LIN {X -206.080,Y 111.413,Z -44.494,A 0.015,B 0.000,C 180.000} C_DIS
LIN {X -204.736,Y 104.947,Z -44.738,A 0.015,B -0.000,C -180.000} C_DIS
LIN {X -198.273,Y 103.588,Z -44.982,A 0.015,B 0.000,C 180.000} C_DIS
LIN {X -194.437,Y 108.964,Z -45.226,A 0.015,B -0.000,C 180.000} C_DIS
LIN {X -197.826,Y 114.632,Z -45.470,A 0.015,B -0.000,C 180.000} C_DIS
LIN {X -204.378,Y 113.799,Z -45.714,A 0.015,B 0.000,C 180.000} C_DIS
LIN {X -206.240,Y 107.463,Z -45.958,A 0.015,B 0.000,C 180.000} C_DIS
LIN {X -201.180,Y 103.218,Z -46.202,A 0.015,B 0.000,C 180.000} C_DIS
LIN {X -195.264,Y 106.152,Z -46.446,A 0.015,B 0.000,C -180.000} C_DIS
LIN {X -195.581,Y 112.749,Z -46.690,A 0.015,B 0.000,C 180.000} C_DIS
LIN {X -201.752,Y 115.101,Z -46.935,A 0.015,B -0.000,C -180.000} C_DIS
LIN {X -206.380,Y 110.390,Z -47.179,A 0.015,B 0.000,C -180.000} C_DIS
LIN {X -203.919,Y 104.262,Z -47.423,A 0.015,B 0.000,C 180.000} C_DIS
LIN {X -197.317,Y 104.061,Z -47.667,A 0.015,B 0.000,C 180.000} C_DIS
LIN {X -194.489,Y 110.029,Z -47.911,A 0.015,B 0.000,C -180.000} C_DIS
LIN {X -198.823,Y 115.012,Z -48.155,A 0.015,B 0.000,C -180.000} C_DIS
LIN {X -205.125,Y 113.038,Z -48.399,A 0.015,B 0.000,C -180.000} C_DIS
LIN {X -205.842,Y 106.473,Z -48.643,A 0.015,B 0.000,C -180.000} C_DIS
LIN {X -200.114,Y 103.185,Z -48.887,A 0.015,B -0.000,C -180.000} C_DIS
LIN {X -194.807,Y 107.116,Z -49.131,A 0.015,B -0.000,C -180.000} C_DIS
LIN {X -196.281,Y 113.554,Z -49.375,A 0.015,B 0.000,C 180.000} C_DIS
LIN {X -202.770,Y 114.782,Z -49.619,A 0.015,B -0.000,C 180.000} C_DIS
LIN {X -206.496,Y 109.330,Z -49.863,A 0.015,B 0.000,C -180.000} C_DIS
LIN {X -202.994,Y 103.731,Z -50.107,A 0.015,B 0.000,C -180.000} C_DIS
LIN {X -196.460,Y 104.696,Z -50.351,A 0.015,B 0.000,C 180.000} C_DIS
LIN {X -194.727,Y 111.069,Z -50.595,A 0.015,B 0.000,C -180.000} C_DIS
LIN {X -199.871,Y 115.211,Z -50.839,A 0.015,B 0.000,C -180.000} C_DIS
LIN {X -205.727,Y 112.158,Z -51.083,A 0.015,B 0.000,C -180.000} C_DIS
LIN {X -205.276,Y 105.569,Z -51.327,A 0.015,B 0.000,C -180.000} C_DIS
LIN {X -199.059,Y 103.341,Z -51.571,A 0.015,B 0.000,C -180.000} C_DIS
LIN {X -194.527,Y 108.145,Z -51.815,A 0.015,B 0.000,C -180.000} C_DIS
LIN {X -197.112,Y 114.223,Z -52.060,A 0.015,B 0.000,C 180.000} C_DIS
LIN {X -203.716,Y 114.289,Z -52.304,A 0.015,B 0.000,C 180.000} C_DIS
LIN {X -206.423,Y 108.265,Z -52.548,A 0.015,B 0.000,C 180.000} C_DIS
LIN {X -201.989,Y 103.371,Z -52.792,A 0.015,B -0.000,C 180.000} C_DIS
LIN {X -195.728,Y 105.472,Z -53.036,A 0.015,B 0.000,C 180.000} C_DIS
LIN {X -195.144,Y 112.051,Z -53.280,A 0.015,B 0.000,C 180.000} C_DIS
LIN {X -200.937,Y 115.222,Z -53.524,A 0.015,B 0.000,C 180.000} C_DIS
LIN {X -206.164,Y 111.185,Z -53.768,A 0.015,B 0.000,C -180.000} C_DIS
LIN {X -204.560,Y 104.778,Z -54.012,A 0.015,B 0.000,C 180.000} C_DIS
LIN {X -198.048,Y 103.681,Z -54.256,A 0.015,B 0.000,C 180.000} C_DIS
LIN {X -194.432,Y 109.208,Z -54.500,A 0.015,B 0.000,C 180.000} C_DIS
CIRC {X -196.756,Y 111.531,Z -54.500,A 0.015,B -0.000,C 180.000},{X -199.080,Y 109.208,Z -54.500,A 0.015,B -0.000,C -180.000} C_DIS
CIRC {X -196.756,Y 106.884,Z -54.500,A 0.015,B 0.000,C -180.000},{X -194.432,Y 109.208,Z -54.500,A 0.015,B 0.000,C -180.000} C_DIS
CIRC {X -193.872,Y 111.256,Z -54.500,A 0.015,B 0.000,C 180.000},{X -192.347,Y 112.733,Z -54.500,A 0.015,B 0.000,C -180.000} C_DIS
CIRC {X -191.132,Y 114.776,Z -54.500,A 0.015,B 0.000,C -180.000},{X -192.330,Y 116.829,Z -54.500,A 0.015,B 0.000,C 180.000} C_DIS
CIRC {X -193.084,Y 117.278,Z -54.500,A 0.015,B 0.000,C -180.000},{X -193.814,Y 117.764,Z -54.500,A 0.015,B -0.000,C 180.000} C_DIS
CIRC {X -196.756,Y 118.696,Z -54.500,A 0.015,B 0.000,C 180.000},{X -199.698,Y 117.764,Z -54.500,A 0.015,B 0.000,C 180.000} C_DIS
CIRC {X -201.103,Y 116.874,Z -54.500,A 0.015,B 0.000,C 180.000},{X -202.588,Y 116.125,Z -54.500,A 0.015,B 0.000,C -180.000} C_DIS
CIRC {X -204.950,Y 114.014,Z -54.500,A 0.015,B -0.000,C 180.000},{X -205.637,Y 110.922,Z -54.500,A 0.015,B 0.000,C -180.000} C_DIS
CIRC {X -205.565,Y 109.268,Z -54.500,A 0.015,B 0.000,C -180.000},{X -205.653,Y 107.615,Z -54.500,A 0.015,B -0.000,C 180.000} C_DIS
CIRC {X -204.998,Y 104.512,Z -54.500,A 0.015,B 0.000,C 180.000},{X -202.663,Y 102.367,Z -54.500,A 0.015,B 0.000,C -180.000} C_DIS
CIRC {X -201.227,Y 101.618,Z -54.500,A 0.015,B 0.000,C -180.000},{X -199.869,Y 100.736,Z -54.500,A 0.015,B 0.000,C -180.000} C_DIS
CIRC {X -196.859,Y 99.736,Z -54.500,A 0.015,B 0.000,C -180.000},{X -193.814,Y 100.624,Z -54.500,A 0.015,B 0.000,C -180.000} C_DIS
CIRC {X -193.079,Y 101.102,Z -54.500,A 0.015,B 0.000,C 180.000},{X -192.334,Y 101.564,Z -54.500,A 0.015,B 0.000,C -180.000} C_DIS
CIRC {X -191.573,Y 101.999,Z -54.500,A 0.015,B 0.000,C -180.000},{X -190.791,Y 102.395,Z -54.500,A 0.015,B 0.000,C -180.000} C_DIS
CIRC {X -188.498,Y 104.537,Z -54.500,A 0.015,B 0.000,C -180.000},{X -187.859,Y 107.610,Z -54.500,A 0.015,B -0.000,C -180.000} C_DIS
CIRC {X -187.947,Y 109.266,Z -54.500,A 0.015,B 0.000,C 180.000},{X -187.875,Y 110.922,Z -54.500,A 0.015,B 0.000,C 180.000} C_DIS
CIRC {X -188.562,Y 114.014,Z -54.500,A 0.015,B 0.000,C 180.000},{X -190.924,Y 116.125,Z -54.500,A 0.015,B 0.000,C 180.000} C_DIS
CIRC {X -191.635,Y 116.461,Z -54.500,A 0.015,B 0.000,C 180.000},{X -192.330,Y 116.829,Z -54.500,A 0.015,B 0.000,C 180.000} C_DIS
LIN {X -192.937,Y 116.991,Z -54.330,A 0.015,B 0.000,C 180.000} C_DIS
LIN {X -193.393,Y 116.912,Z -53.865,A 0.015,B 0.000,C -180.000} C_DIS
LIN {X -193.548,Y 116.842,Z -53.230,A 0.015,B 0.000,C 180.000} C_DIS
$VEL.CP = 1.00000
LIN {X -193.548,Y 116.842,Z 11.000,A 0.015,B 0.000,C 180.000} C_DIS
$VEL.CP = 1.00000
LIN {X -195.993,Y 9.529,Z 11.000,A 0.015,B 0.000,C -180.000} C_DIS
$VEL.CP = 1.00000
LIN {X -195.993,Y 9.529,Z -32.731,A 0.015,B 0.000,C 180.000} C_DIS
$VEL.CP = 0.10000
LIN {X -196.154,Y 9.547,Z -33.353,A 0.015,B 0.000,C 180.000} C_DIS
LIN {X -196.600,Y 9.576,Z -33.816,A 0.015,B 0.000,C 180.000} C_DIS
LIN {X -197.216,Y 9.560,Z -34.000,A 0.015,B -0.000,C -180.000} C_DIS
LIN {X -202.453,Y 5.536,Z -34.244,A 0.015,B 0.000,C -180.000} C_DIS
LIN {X -200.864,Y -0.874,Z -34.488,A 0.015,B 0.000,C 180.000} C_DIS
LIN {X -194.354,Y -1.988,Z -34.732,A 0.015,B 0.000,C 180.000} C_DIS
LIN {X -190.726,Y 3.530,Z -34.976,A 0.015,B 0.000,C 180.000} C_DIS
LIN {X -194.327,Y 9.066,Z -35.220,A 0.015,B 0.000,C 180.000} C_DIS
LIN {X -200.842,Y 7.985,Z -35.464,A 0.015,B -0.000,C -180.000} C_DIS
LIN {X -202.462,Y 1.582,Z -35.708,A 0.015,B 0.000,C -180.000} C_DIS
LIN {X -197.245,Y -2.468,Z -35.952,A 0.015,B -0.000,C 180.000} C_DIS
LIN {X -191.445,Y 0.689,Z -36.196,A 0.015,B -0.000,C 180.000} C_DIS
LIN {X -192.012,Y 7.269,Z -36.440,A 0.015,B 0.000,C -180.000} C_DIS
LIN {X -198.268,Y 9.386,Z -36.685,A 0.015,B 0.000,C 180.000} C_DIS
LIN {X -202.714,Y 4.502,Z -36.929,A 0.015,B 0.000,C -180.000} C_DIS
LIN {X -200.022,Y -1.528,Z -37.173,A 0.015,B 0.000,C -180.000} C_DIS
LIN {X -193.417,Y -1.478,Z -37.417,A 0.015,B 0.000,C 180.000} C_DIS
LIN {X -190.817,Y 4.593,Z -37.661,A 0.015,B 0.000,C -180.000} C_DIS
LIN {X -195.338,Y 9.408,Z -37.905,A 0.015,B -0.000,C 180.000} C_DIS
LIN {X -201.560,Y 7.196,Z -38.149,A 0.015,B 0.000,C -180.000} C_DIS
LIN {X -202.027,Y 0.608,Z -38.393,A 0.015,B 0.000,C -180.000} C_DIS
LIN {X -196.179,Y -2.459,Z -38.637,A 0.015,B 0.000,C -180.000} C_DIS
LIN {X -191.025,Y 1.670,Z -38.881,A 0.015,B 0.000,C 180.000} C_DIS
LIN {X -192.742,Y 8.047,Z -39.125,A 0.015,B 0.000,C 180.000} C_DIS
LIN {X -199.273,Y 9.028,Z -39.369,A 0.015,B 0.000,C 180.000} C_DIS
LIN {X -202.790,Y 3.438,Z -39.613,A 0.015,B 0.000,C -180.000} C_DIS
LIN {X -199.077,Y -2.024,Z -39.857,A 0.015,B 0.000,C 180.000} C_DIS
LIN {X -192.585,Y -0.811,Z -40.101,A 0.015,B -0.000,C -180.000} C_DIS
LIN {X -191.095,Y 5.623,Z -40.345,A 0.015,B 0.000,C -180.000} C_DIS
LIN {X -196.392,Y 9.567,Z -40.589,A 0.015,B 0.000,C -180.000} C_DIS
LIN {X -202.128,Y 6.293,Z -40.833,A 0.015,B -0.000,C -180.000} C_DIS
LIN {X -201.428,Y -0.274,Z -41.077,A 0.015,B 0.000,C -180.000} C_DIS
LIN {X -195.130,Y -2.263,Z -41.321,A 0.015,B 0.000,C -180.000} C_DIS
LIN {X -190.784,Y 2.709,Z -41.565,A 0.015,B 0.000,C -180.000} C_DIS
LIN {X -193.598,Y 8.684,Z -41.810,A 0.015,B -0.000,C 180.000} C_DIS
LIN {X -200.200,Y 8.500,Z -42.054,A 0.015,B 0.000,C -180.000} C_DIS
LIN {X -202.677,Y 2.377,Z -42.298,A 0.015,B -0.000,C -180.000} C_DIS
LIN {X -198.060,Y -2.345,Z -42.542,A 0.015,B 0.000,C 180.000} C_DIS
LIN {X -191.883,Y -0.008,Z -42.786,A 0.015,B 0.000,C -180.000} C_DIS
LIN {X -191.549,Y 6.588,Z -43.030,A 0.015,B 0.000,C -180.000} C_DIS
LIN {X -197.459,Y 9.537,Z -43.274,A 0.015,B -0.000,C 180.000} C_DIS
LIN {X -202.528,Y 5.304,Z -43.518,A 0.015,B 0.000,C 180.000} C_DIS
LIN {X -200.682,Y -1.037,Z -43.762,A 0.015,B 0.000,C -180.000} C_DIS
LIN {X -194.133,Y -1.886,Z -44.006,A 0.015,B 0.000,C 180.000} C_DIS
LIN {X -190.730,Y 3.774,Z -44.250,A 0.015,B 0.000,C 180.000} C_DIS
LIN {X -194.552,Y 9.160,Z -44.494,A 0.015,B 0.000,C 180.000} C_DIS
LIN {X -201.018,Y 7.816,Z -44.738,A 0.015,B 0.000,C 180.000} C_DIS
LIN {X -202.378,Y 1.353,Z -44.982,A 0.015,B -0.000,C -180.000} C_DIS
LIN {X -197.002,Y -2.482,Z -45.226,A 0.015,B 0.000,C -180.000} C_DIS
LIN {X -191.333,Y 0.906,Z -45.470,A 0.015,B 0.000,C -180.000} C_DIS
LIN {X -192.167,Y 7.458,Z -45.714,A 0.015,B 0.000,C -180.000} C_DIS
LIN {X -198.503,Y 9.320,Z -45.958,A 0.015,B 0.000,C -180.000} C_DIS
LIN {X -202.748,Y 4.261,Z -46.202,A 0.015,B -0.000,C -180.000} C_DIS
LIN {X -199.814,Y -1.656,Z -46.446,A 0.015,B -0.000,C -180.000} C_DIS
LIN {X -193.217,Y -1.339,Z -46.690,A 0.015,B -0.000,C 180.000} C_DIS
LIN {X -190.865,Y 4.832,Z -46.935,A 0.015,B -0.000,C -180.000} C_DIS
LIN {X -195.576,Y 9.461,Z -47.179,A 0.015,B -0.000,C -180.000} C_DIS
LIN {X -201.704,Y 6.999,Z -47.423,A 0.015,B 0.000,C -180.000} C_DIS
LIN {X -201.904,Y 0.398,Z -47.667,A 0.015,B 0.000,C 180.000} C_DIS
LIN {X -195.937,Y -2.431,Z -47.911,A 0.015,B -0.000,C 180.000} C_DIS
LIN {X -190.953,Y 1.903,Z -48.155,A 0.015,B 0.000,C -180.000} C_DIS
LIN {X -192.928,Y 8.206,Z -48.399,A 0.015,B 0.000,C -180.000} C_DIS
LIN {X -199.493,Y 8.922,Z -48.643,A 0.015,B 0.000,C -180.000} C_DIS
LIN {X -202.780,Y 3.194,Z -48.887,A 0.015,B 0.000,C 180.000} C_DIS
LIN {X -198.850,Y -2.113,Z -49.131,A 0.015,B -0.000,C 180.000} C_DIS
